LIN {X 0,Y 300.926,Z 371.519,A -85,B 0,C 180,E1 -19127.821,E2 -19127.821} C_VEL
LIN {X 0,Y 293.445,Z 384.523,A -85,B 0,C 180,E1 -19129.259,E2 -19129.259} C_VEL
LIN {X 0,Y 285.391,Z 397.595,A -85,B 0,C 180,E1 -19131.1,E2 -19131.1} C_VEL
LIN {X 0,Y 277.927,Z 408.98,A -85,B 0,C 180,E1 -19133.089,E2 -19133.089} C_VEL
LIN {X 0,Y 270.199,Z 420.219,A -85,B 0,C 180,E1 -19135.547,E2 -19135.547} C_VEL
LIN {X 0,Y 262.579,Z 430.974,A -85,B 0,C 180,E1 -19138.539,E2 -19138.539} C_VEL
LIN {X 0,Y 256.104,Z 439.853,A -85,B 0,C 180,E1 -19141.687,E2 -19141.687} C_VEL
LIN {X 0,Y 251.781,Z 445.833,A -85,B 0,C 180,E1 -19144.364,E2 -19144.364} C_VEL
LIN {X 0,Y 247.717,Z 451.471,A -85,B 0,C 180,E1 -19147.48,E2 -19147.48} C_VEL
LIN {X 0,Y 245.217,Z 454.914,A -85,B 0,C 180,E1 -19149.884,E2 -19149.884} C_VEL
LIN {X 0,Y 243.007,Z 458.084,A -85,B 0,C 180,E1 -19152.628,E2 -19152.628} C_VEL
LIN {X 0,Y 241.525,Z 462.948,A -85,B 0,C 180,E1 -19155.68,E2 -19155.68} C_VEL
LIN {X 0,Y 240.587,Z 466.054,A -85,B 0,C 180,E1 -19158.201,E2 -19158.201} C_VEL
LIN {X 0,Y 240.006,Z 469.152,A -85,B 0,C 180,E1 -19161.581,E2 -19161.581} C_VEL
LIN {X 0,Y 239.791,Z 471.129,A -85,B 0,C 180,E1 -19165.2,E2 -19165.2} C_VEL
LIN {X 0,Y 239.847,Z 471.756,A -85,B 0,C 180,E1 -19168.321,E2 -19168.321} C_VEL
LIN {X 0,Y 239.895,Z 471.645,A -85,B 0,C 180,E1 -19170,E2 -19170} C_VEL
LIN {X 0,Y 239.802,Z 470.52,A -85,B 0,C 180,E1 -19173.36,E2 -19173.36} C_VEL
LIN {X 0,Y 239.871,Z 468.169,A -85,B 0,C 180,E1 -19176.73,E2 -19176.73} C_VEL
LIN {X 0,Y 240.17,Z 464.526,A -85,B 0,C 180,E1 -19180.112,E2 -19180.112} C_VEL
LIN {X 0,Y 241.011,Z 459.793,A -85,B 0,C 180,E1 -19183.491,E2 -19183.491} C_VEL
LIN {X 0,Y 242.828,Z 456.84,A -85,B 0,C 180,E1 -19187.237,E2 -19187.237} C_VEL
LIN {X 0,Y 245.914,Z 452.461,A -85,B 0,C 180,E1 -19190.931,E2 -19190.931} C_VEL
LIN {X 0,Y 249.577,Z 447.385,A -85,B 0,C 180,E1 -19194.099,E2 -19194.099} C_VEL
LIN {X 0,Y 254.007,Z 441.145,A -85,B 0,C 180,E1 -19197.163,E2 -19197.163} C_VEL
LIN {X 0,Y 259.413,Z 433.669,A -85,B 0,C 180,E1 -19200.079,E2 -19200.079} C_VEL
LIN {X 0,Y 266.658,Z 423.616,A -85,B 0,C 180,E1 -19203.154,E2 -19203.154} C_VEL
LIN {X 0,Y 274.949,Z 411.661,A -85,B 0,C 180,E1 -19206.009,E2 -19206.009} C_VEL
LIN {X 0,Y 283.218,Z 399.07,A -85,B 0,C 180,E1 -19208.343,E2 -19208.343} C_VEL
LIN {X 0,Y 292.329,Z 384.265,A -85,B 0,C 180,E1 -19210.475,E2 -19210.475} C_VEL
LIN {X 0,Y 300.405,Z 370.081,A -85,B 0,C 180,E1 -19212.043,E2 -19212.043} C_VEL
LIN {X 0,Y 308.472,Z 354.464,A -85,B 0,C 180,E1 -19213.364,E2 -19213.364} C_VEL
LIN {X 0,Y 315.333,Z 339.378,A -85,B 0,C 180,E1 -19214.338,E2 -19214.338} C_VEL
LIN {X 0,Y 322.129,Z 322.096,A -85,B 0,C 180,E1 -19215.191,E2 -19215.191} C_VEL
LIN {X 0,Y 323.521,Z 318.179,A -85,B 0,C 180,E1 -19215.353,E2 -19215.353} C_VEL
LIN {X 0,Y 323.563,Z 317.976,A -85,B 0,C 180,E1 -19215.539,E2 -19215.539} C_VEL
LIN {X 0,Y 317.653,Z 333.405,A -85,B 0,C 180,E1 -19216.478,E2 -19216.478} C_VEL
LIN {X 0,Y 310.672,Z 348.818,A -85,B 0,C 180,E1 -19217.701,E2 -19217.701} C_VEL
LIN {X 0,Y 302.844,Z 363.944,A -85,B 0,C 180,E1 -19219.256,E2 -19219.256} C_VEL
LIN {X 0,Y 295.502,Z 376.592,A -85,B 0,C 180,E1 -19220.931,E2 -19220.931} C_VEL
LIN {X 0,Y 287.997,Z 388.352,A -85,B 0,C 180,E1 -19222.845,E2 -19222.845} C_VEL
LIN {X 0,Y 280.124,Z 399.752,A -85,B 0,C 180,E1 -19225.196,E2 -19225.196} C_VEL
LIN {X 0,Y 273.695,Z 408.358,A -85,B 0,C 180,E1 -19227.368,E2 -19227.368} C_VEL
LIN {X 0,Y 267.129,Z 416.621,A -85,B 0,C 180,E1 -19230.009,E2 -19230.009} C_VEL
LIN {X 0,Y 261.275,Z 423.494,A -85,B 0,C 180,E1 -19232.789,E2 -19232.789} C_VEL
LIN {X 0,Y 256.163,Z 429.083,A -85,B 0,C 180,E1 -19235.699,E2 -19235.699} C_VEL
LIN {X 0,Y 251.642,Z 433.523,A -85,B 0,C 180,E1 -19238.712,E2 -19238.712} C_VEL
LIN {X 0,Y 248.08,Z 436.727,A -85,B 0,C 180,E1 -19241.843,E2 -19241.843} C_VEL
LIN {X 0,Y 245.226,Z 438.819,A -85,B 0,C 180,E1 -19245.053,E2 -19245.053} C_VEL
LIN {X 0,Y 243.131,Z 439.825,A -85,B 0,C 180,E1 -19248.326,E2 -19248.326} C_VEL
LIN {X 0,Y 241.522,Z 439.746,A -85,B 0,C 180,E1 -19251.635,E2 -19251.635} C_VEL
LIN {X 0,Y 240.629,Z 438.526,A -85,B 0,C 180,E1 -19254.974,E2 -19254.974} C_VEL
LIN {X 0,Y 240.193,Z 436.107,A -85,B 0,C 180,E1 -19258.324,E2 -19258.324} C_VEL
LIN {X 0,Y 240.07,Z 432.433,A -85,B 0,C 180,E1 -19261.678,E2 -19261.678} C_VEL
LIN {X 0,Y 240.095,Z 427.408,A -85,B 0,C 180,E1 -19265.038,E2 -19265.038} C_VEL
LIN {X 0,Y 240.395,Z 422.656,A -85,B 0,C 180,E1 -19267.56,E2 -19267.56} C_VEL
LIN {X 0,Y 240.816,Z 415.933,A -85,B 0,C 180,E1 -19270.51,E2 -19270.51} C_VEL
LIN {X 0,Y 241.661,Z 407.787,A -85,B 0,C 180,E1 -19273.454,E2 -19273.454} C_VEL
LIN {X 0,Y 242.58,Z 399.463,A -85,B 0,C 180,E1 -19275.976,E2 -19275.976} C_VEL
LIN {X 0,Y 244.039,Z 387.89,A -85,B 0,C 180,E1 -19278.905,E2 -19278.905} C_VEL
LIN {X 0,Y 245.852,Z 374.969,A -85,B 0,C 180,E1 -19281.596,E2 -19281.596} C_VEL
LIN {X 0,Y 247.613,Z 361.872,A -85,B 0,C 180,E1 -19283.858,E2 -19283.858} C_VEL
LIN {X 0,Y 249.407,Z 348.878,A -85,B 0,C 180,E1 -19285.72,E2 -19285.72} C_VEL
LIN {X 0,Y 251.213,Z 333.884,A -85,B 0,C 180,E1 -19287.492,E2 -19287.492} C_VEL
LIN {X 0,Y 252.942,Z 318.105,A -85,B 0,C 180,E1 -19288.98,E2 -19288.98} C_VEL
LIN {X 0,Y 254.311,Z 301.663,A -85,B 0,C 180,E1 -19290.174,E2 -19290.174} C_VEL
LIN {X 0,Y 255.554,Z 284.029,A -85,B 0,C 180,E1 -19291.099,E2 -19291.099} C_VEL
LIN {X 0,Y 261.943,Z 188.853,A -85,B 0,C 180,E1 -19295.144,E2 -19295.144} C_VEL
LIN {X 0,Y 247.071,Z 153.283,A -85,B 0,C 180,E1 -19298.227,E2 -19298.227} C_VEL
LIN {X 0,Y 242.059,Z 141.421,A -85,B 0,C 180,E1 -19299.345,E2 -19299.345} C_VEL
LIN {X 0,Y 241.982,Z 140.968,A -85,B 0,C 180,E1 -19299.451,E2 -19299.451} C_VEL
LIN {X 0,Y 241.902,Z 140.961,A -85,B 0,C 180,E1 -19304.21,E2 -19304.21} C_VEL
LIN {X 0,Y 241.91,Z 140.944,A -85,B 0,C 180,E1 -19308.072,E2 -19308.072} C_VEL
LIN {X 0,Y 241.985,Z 140.951,A -85,B 0,C 180,E1 -19312.417,E2 -19312.417} C_VEL
LIN {X 0,Y 241.982,Z 140.957,A -85,B 0,C 180,E1 -19316.508,E2 -19316.508} C_VEL
LIN {X 0,Y 241.979,Z 140.944,A -85,B 0,C 180,E1 -19320.613,E2 -19320.613} C_VEL
LIN {X 0,Y 241.999,Z 140.959,A -85,B 0,C 180,E1 -19324.197,E2 -19324.197} C_VEL
LIN {X 0,Y 241.98,Z 141.039,A -85,B 0,C 180,E1 -19327.592,E2 -19327.592} C_VEL
LIN {X 0,Y 242.401,Z 142.66,A -85,B 0,C 180,E1 -19328.094,E2 -19328.094} C_VEL
LIN {X 0,Y 244.421,Z 146.942,A -85,B 0,C 180,E1 -19329.518,E2 -19329.518} C_VEL
LIN {X 0,Y 252.986,Z 160.771,A -85,B 0,C 180,E1 -19331.795,E2 -19331.795} C_VEL
LIN {X 0,Y 261.458,Z 175.871,A -85,B 0,C 180,E1 -19333.915,E2 -19333.915} C_VEL
LIN {X 0,Y 269.699,Z 192.53,A -85,B 0,C 180,E1 -19335.885,E2 -19335.885} C_VEL
LIN {X 0,Y 275.294,Z 205.581,A -85,B 0,C 180,E1 -19337.192,E2 -19337.192} C_VEL
LIN {X 0,Y 269.954,Z 313.697,A -85,B 0,C 180,E1 -19340.021,E2 -19340.021} C_VEL
LIN {X 0,Y 268.503,Z 329.395,A -85,B 0,C 180,E1 -19340.68,E2 -19340.68} C_VEL
LIN {X 0,Y 266.769,Z 343.814,A -85,B 0,C 180,E1 -19341.573,E2 -19341.573} C_VEL
LIN {X 0,Y 264.506,Z 358.15,A -85,B 0,C 180,E1 -19342.749,E2 -19342.749} C_VEL
LIN {X 0,Y 261.843,Z 371.771,A -85,B 0,C 180,E1 -19344.172,E2 -19344.172} C_VEL
LIN {X 0,Y 258.88,Z 385.03,A -85,B 0,C 180,E1 -19345.913,E2 -19345.913} C_VEL
LIN {X 0,Y 255.933,Z 396.923,A -85,B 0,C 180,E1 -19347.836,E2 -19347.836} C_VEL
LIN {X 0,Y 252.994,Z 407.937,A -85,B 0,C 180,E1 -19350,E2 -19350} C_VEL
LIN {X 0,Y 250.073,Z 418.104,A -85,B 0,C 180,E1 -19352.416,E2 -19352.416} C_VEL
LIN {X 0,Y 247.562,Z 426.707,A -85,B 0,C 180,E1 -19354.886,E2 -19354.886} C_VEL
LIN {X 0,Y 245.125,Z 435.113,A -85,B 0,C 180,E1 -19357.827,E2 -19357.827} C_VEL
LIN {X 0,Y 243.215,Z 441.844,A -85,B 0,C 180,E1 -19360.74,E2 -19360.74} C_VEL
LIN {X 0,Y 241.894,Z 446.911,A -85,B 0,C 180,E1 -19363.44,E2 -19363.44} C_VEL
LIN {X 0,Y 240.686,Z 452.108,A -85,B 0,C 180,E1 -19366.978,E2 -19366.978} C_VEL
LIN {X 0,Y 239.819,Z 455.891,A -85,B 0,C 180,E1 -19370.589,E2 -19370.589} C_VEL
LIN {X 0,Y 239.462,Z 458.272,A -85,B 0,C 180,E1 -19374.261,E2 -19374.261} C_VEL
LIN {X 0,Y 239.408,Z 459.268,A -85,B 0,C 180,E1 -19378.014,E2 -19378.014} C_VEL
LIN {X 0,Y 239.683,Z 458.815,A -85,B 0,C 180,E1 -19381.857,E2 -19381.857} C_VEL
LIN {X 0,Y 240.458,Z 456.825,A -85,B 0,C 180,E1 -19385.771,E2 -19385.771} C_VEL
LIN {X 0,Y 241.248,Z 454.814,A -85,B 0,C 180,E1 -19388.134,E2 -19388.134} C_VEL
LIN {X 0,Y 242.842,Z 450.587,A -85,B 0,C 180,E1 -19391.731,E2 -19391.731} C_VEL
LIN {X 0,Y 244.71,Z 445.781,A -85,B 0,C 180,E1 -19394.779,E2 -19394.779} C_VEL
LIN {X 0,Y 247.458,Z 438.873,A -85,B 0,C 180,E1 -19398.147,E2 -19398.147} C_VEL
LIN {X 0,Y 250.65,Z 431.232,A -85,B 0,C 180,E1 -19401.086,E2 -19401.086} C_VEL
LIN {X 0,Y 254.215,Z 422.206,A -85,B 0,C 180,E1 -19403.888,E2 -19403.888} C_VEL
LIN {X 0,Y 258.092,Z 411.8,A -85,B 0,C 180,E1 -19406.497,E2 -19406.497} C_VEL
LIN {X 0,Y 262.065,Z 400.682,A -85,B 0,C 180,E1 -19408.74,E2 -19408.74} C_VEL
LIN {X 0,Y 265.88,Z 388.642,A -85,B 0,C 180,E1 -19410.726,E2 -19410.726} C_VEL
LIN {X 0,Y 269.557,Z 375.766,A -85,B 0,C 180,E1 -19412.432,E2 -19412.432} C_VEL
LIN {X 0,Y 270.028,Z 373.954,A -85,B 0,C 180,E1 -19412.644,E2 -19412.644} C_VEL
LIN {X 0,Y 269.51,Z 373.561,A -85,B 0,C 180,E1 -19412.806,E2 -19412.806} C_VEL
LIN {X 0,Y 260.352,Z 374.742,A -85,B 0,C 180,E1 -19414.411,E2 -19414.411} C_VEL
LIN {X 0,Y 254.665,Z 374.937,A -85,B 0,C 180,E1 -19415.603,E2 -19415.603} C_VEL
LIN {X 0,Y 247.238,Z 374.53,A -85,B 0,C 180,E1 -19417.433,E2 -19417.433} C_VEL
LIN {X 0,Y 246.295,Z 373.126,A -85,B 0,C 180,E1 -19418.005,E2 -19418.005} C_VEL
LIN {X 0,Y 244.695,Z 384.518,A -85,B 0,C 180,E1 -19420.276,E2 -19420.276} C_VEL
LIN {X 0,Y 243.165,Z 395.558,A -85,B 0,C 180,E1 -19422.892,E2 -19422.892} C_VEL
LIN {X 0,Y 242.388,Z 402.645,A -85,B 0,C 180,E1 -19424.843,E2 -19424.843} C_VEL
LIN {X 0,Y 241.37,Z 406.257,A -85,B 0,C 180,E1 -19425.92,E2 -19425.92} C_VEL
LIN {X 0,Y 237.891,Z 411.633,A -85,B 0,C 180,E1 -19427.73,E2 -19427.73} C_VEL
LIN {X 0,Y 234.449,Z 416.584,A -85,B 0,C 180,E1 -19429.662,E2 -19429.662} C_VEL
LIN {X 0,Y 233.518,Z 419.483,A -85,B 0,C 180,E1 -19430.91,E2 -19430.91} C_VEL
LIN {X 0,Y 233.1,Z 426.282,A -85,B 0,C 180,E1 -19434.244,E2 -19434.244} C_VEL
LIN {X 0,Y 233.038,Z 431.403,A -85,B 0,C 180,E1 -19437.407,E2 -19437.407} C_VEL
LIN {X 0,Y 233.02,Z 434.736,A -85,B 0,C 180,E1 -19439.999,E2 -19439.999} C_VEL
LIN {X 0,Y 233.386,Z 438.017,A -85,B 0,C 180,E1 -19443.452,E2 -19443.452} C_VEL
LIN {X 0,Y 233.983,Z 440.115,A -85,B 0,C 180,E1 -19446.9,E2 -19446.9} C_VEL
LIN {X 0,Y 235.344,Z 441.087,A -85,B 0,C 180,E1 -19450.321,E2 -19450.321} C_VEL
LIN {X 0,Y 237.262,Z 440.964,A -85,B 0,C 180,E1 -19453.707,E2 -19453.707} C_VEL
LIN {X 0,Y 239.772,Z 439.723,A -85,B 0,C 180,E1 -19457.044,E2 -19457.044} C_VEL
LIN {X 0,Y 243.236,Z 437.397,A -85,B 0,C 180,E1 -19460.287,E2 -19460.287} C_VEL
LIN {X 0,Y 247.434,Z 434.005,A -85,B 0,C 180,E1 -19463.431,E2 -19463.431} C_VEL
LIN {X 0,Y 252.482,Z 429.476,A -85,B 0,C 180,E1 -19466.447,E2 -19466.447} C_VEL
LIN {X 0,Y 259.22,Z 422.76,A -85,B 0,C 180,E1 -19469.757,E2 -19469.757} C_VEL
LIN {X 0,Y 266.506,Z 414.81,A -85,B 0,C 180,E1 -19472.724,E2 -19472.724} C_VEL
LIN {X 0,Y 274.914,Z 404.883,A -85,B 0,C 180,E1 -19475.562,E2 -19475.562} C_VEL
LIN {X 0,Y 283.036,Z 394.461,A -85,B 0,C 180,E1 -19477.92,E2 -19477.92} C_VEL
LIN {X 0,Y 291.952,Z 382.057,A -85,B 0,C 180,E1 -19480.086,E2 -19480.086} C_VEL
LIN {X 0,Y 300.223,Z 369.287,A -85,B 0,C 180,E1 -19481.848,E2 -19481.848} C_VEL
LIN {X 0,Y 307.069,Z 357.731,A -85,B 0,C 180,E1 -19483.138,E2 -19483.138} C_VEL
LIN {X 0,Y 312.933,Z 346.743,A -85,B 0,C 180,E1 -19484.124,E2 -19484.124} C_VEL
LIN {X 0,Y 313.613,Z 345.475,A -85,B 0,C 180,E1 -19484.431,E2 -19484.431} C_VEL
LIN {X 0,Y 305.164,Z 361.795,A -85,B 0,C 180,E1 -19485.556,E2 -19485.556} C_VEL
LIN {X 0,Y 296.187,Z 377.189,A -85,B 0,C 180,E1 -19486.985,E2 -19486.985} C_VEL
LIN {X 0,Y 287.36,Z 391.028,A -85,B 0,C 180,E1 -19488.674,E2 -19488.674} C_VEL
LIN {X 0,Y 278.033,Z 404.592,A -85,B 0,C 180,E1 -19490.807,E2 -19490.807} C_VEL
LIN {X 0,Y 269.529,Z 416.205,A -85,B 0,C 180,E1 -19493.15,E2 -19493.15} C_VEL
LIN {X 0,Y 261.948,Z 426.171,A -85,B 0,C 180,E1 -19495.707,E2 -19495.707} C_VEL
LIN {X 0,Y 255.106,Z 434.753,A -85,B 0,C 180,E1 -19498.437,E2 -19498.437} C_VEL
LIN {X 0,Y 249.184,Z 442.052,A -85,B 0,C 180,E1 -19501.349,E2 -19501.349} C_VEL
LIN {X 0,Y 244.279,Z 448.164,A -85,B 0,C 180,E1 -19504.434,E2 -19504.434} C_VEL
LIN {X 0,Y 240.247,Z 453.191,A -85,B 0,C 180,E1 -19507.648,E2 -19507.648} C_VEL
LIN {X 0,Y 235.865,Z 459.03,A -85,B 0,C 180,E1 -19512.664,E2 -19512.664} C_VEL
LIN {X 0,Y 234.232,Z 464.005,A -85,B 0,C 180,E1 -19516.111,E2 -19516.111} C_VEL
LIN {X 0,Y 233.179,Z 467.672,A -85,B 0,C 180,E1 -19519.581,E2 -19519.581} C_VEL
LIN {X 0,Y 232.79,Z 470.12,A -85,B 0,C 180,E1 -19523.064,E2 -19523.064} C_VEL
LIN {X 0,Y 232.682,Z 471.387,A -85,B 0,C 180,E1 -19526.537,E2 -19526.537} C_VEL
LIN {X 0,Y 232.806,Z 471.448,A -85,B 0,C 180,E1 -19530,E2 -19530} C_VEL
LIN {X 0,Y 232.708,Z 470.282,A -85,B 0,C 180,E1 -19533.463,E2 -19533.463} C_VEL
LIN {X 0,Y 232.785,Z 467.887,A -85,B 0,C 180,E1 -19536.936,E2 -19536.936} C_VEL
LIN {X 0,Y 233.116,Z 464.197,A -85,B 0,C 180,E1 -19540.422,E2 -19540.422} C_VEL
LIN {X 0,Y 233.959,Z 459.718,A -85,B 0,C 180,E1 -19543.684,E2 -19543.684} C_VEL
LIN {X 0,Y 235.834,Z 457.13,A -85,B 0,C 180,E1 -19547.52,E2 -19547.52} C_VEL
LIN {X 0,Y 239.29,Z 452.881,A -85,B 0,C 180,E1 -19551.539,E2 -19551.539} C_VEL
LIN {X 0,Y 243.126,Z 448.136,A -85,B 0,C 180,E1 -19554.781,E2 -19554.781} C_VEL
LIN {X 0,Y 247.804,Z 442.286,A -85,B 0,C 180,E1 -19557.902,E2 -19557.902} C_VEL
LIN {X 0,Y 253.449,Z 435.245,A -85,B 0,C 180,E1 -19560.864,E2 -19560.864} C_VEL
LIN {X 0,Y 260.093,Z 426.873,A -85,B 0,C 180,E1 -19563.637,E2 -19563.637} C_VEL
LIN {X 0,Y 267.58,Z 417.126,A -85,B 0,C 180,E1 -19566.225,E2 -19566.225} C_VEL
LIN {X 0,Y 274.794,Z 407.302,A -85,B 0,C 180,E1 -19568.331,E2 -19568.331} C_VEL
LIN {X 0,Y 282.677,Z 396.052,A -85,B 0,C 180,E1 -19570.272,E2 -19570.272} C_VEL
LIN {X 0,Y 291.787,Z 382.13,A -85,B 0,C 180,E1 -19572.175,E2 -19572.175} C_VEL
LIN {X 0,Y 300.368,Z 367.891,A -85,B 0,C 180,E1 -19573.649,E2 -19573.649} C_VEL
LIN {X 0,Y 308.765,Z 352.317,A -85,B 0,C 180,E1 -19574.879,E2 -19574.879} C_VEL
LIN {X 0,Y 312.951,Z 343.745,A -85,B 0,C 180,E1 -19575.419,E2 -19575.419} C_VEL
LIN {X 0,Y 313.381,Z 342.678,A -85,B 0,C 180,E1 -19575.791,E2 -19575.791} C_VEL
LIN {X 0,Y 306.429,Z 356.216,A -85,B 0,C 180,E1 -19576.975,E2 -19576.975} C_VEL
LIN {X 0,Y 298.992,Z 369.068,A -85,B 0,C 180,E1 -19578.392,E2 -19578.392} C_VEL
LIN {X 0,Y 289.686,Z 383.476,A -85,B 0,C 180,E1 -19580.444,E2 -19580.444} C_VEL
LIN {X 0,Y 282.043,Z 394.205,A -85,B 0,C 180,E1 -19582.375,E2 -19582.375} C_VEL
LIN {X 0,Y 272.96,Z 405.879,A -85,B 0,C 180,E1 -19585.049,E2 -19585.049} C_VEL
LIN {X 0,Y 265.624,Z 414.565,A -85,B 0,C 180,E1 -19587.603,E2 -19587.603} C_VEL
LIN {X 0,Y 258.219,Z 422.674,A -85,B 0,C 180,E1 -19590.666,E2 -19590.666} C_VEL
LIN {X 0,Y 251.229,Z 429.713,A -85,B 0,C 180,E1 -19594.304,E2 -19594.304} C_VEL
LIN {X 0,Y 247.459,Z 433.067,A -85,B 0,C 180,E1 -19596.572,E2 -19596.572} C_VEL
LIN {X 0,Y 243.172,Z 436.579,A -85,B 0,C 180,E1 -19599.708,E2 -19599.708} C_VEL
LIN {X 0,Y 239.77,Z 438.959,A -85,B 0,C 180,E1 -19602.956,E2 -19602.956} C_VEL
LIN {X 0,Y 237.231,Z 440.253,A -85,B 0,C 180,E1 -19606.291,E2 -19606.291} C_VEL
LIN {X 0,Y 235.256,Z 440.439,A -85,B 0,C 180,E1 -19609.675,E2 -19609.675} C_VEL
LIN {X 0,Y 233.942,Z 439.523,A -85,B 0,C 180,E1 -19613.099,E2 -19613.099} C_VEL
LIN {X 0,Y 233.335,Z 437.473,A -85,B 0,C 180,E1 -19616.547,E2 -19616.547} C_VEL
LIN {X 0,Y 233.012,Z 434.229,A -85,B 0,C 180,E1 -19620.001,E2 -19620.001} C_VEL
LIN {X 0,Y 232.99,Z 429.672,A -85,B 0,C 180,E1 -19623.459,E2 -19623.459} C_VEL
LIN {X 0,Y 233.218,Z 423.655,A -85,B 0,C 180,E1 -19626.924,E2 -19626.924} C_VEL
LIN {X 0,Y 233.659,Z 417.081,A -85,B 0,C 180,E1 -19629.96,E2 -19629.96} C_VEL
LIN {X 0,Y 234.399,Z 409.058,A -85,B 0,C 180,E1 -19632.996,E2 -19632.996} C_VEL
LIN {X 0,Y 235.309,Z 400.854,A -85,B 0,C 180,E1 -19635.594,E2 -19635.594} C_VEL
LIN {X 0,Y 236.606,Z 390.774,A -85,B 0,C 180,E1 -19638.306,E2 -19638.306} C_VEL
LIN {X 0,Y 238.205,Z 378.995,A -85,B 0,C 180,E1 -19640.962,E2 -19640.962} C_VEL
LIN {X 0,Y 239.973,Z 366.61,A -85,B 0,C 180,E1 -19643.29,E2 -19643.29} C_VEL
LIN {X 0,Y 241.849,Z 353.276,A -85,B 0,C 180,E1 -19645.381,E2 -19645.381} C_VEL
LIN {X 0,Y 243.652,Z 338.78,A -85,B 0,C 180,E1 -19647.252,E2 -19647.252} C_VEL
LIN {X 0,Y 245.472,Z 322.964,A -85,B 0,C 180,E1 -19648.891,E2 -19648.891} C_VEL
LIN {X 0,Y 247.014,Z 306.649,A -85,B 0,C 180,E1 -19650.215,E2 -19650.215} C_VEL
LIN {X 0,Y 248.289,Z 289.889,A -85,B 0,C 180,E1 -19651.222,E2 -19651.222} C_VEL
LIN {X 0,Y 255.155,Z 190.478,A -85,B 0,C 180,E1 -19655.633,E2 -19655.633} C_VEL
LIN {X 0,Y 240.998,Z 156.526,A -85,B 0,C 180,E1 -19658.644,E2 -19658.644} C_VEL
LIN {X 0,Y 234.996,Z 142.381,A -85,B 0,C 180,E1 -19660.021,E2 -19660.021} C_VEL
LIN {X 0,Y 234.92,Z 141.848,A -85,B 0,C 180,E1 -19660.074,E2 -19660.074} C_VEL
LIN {X 0,Y 234.869,Z 141.838,A -85,B 0,C 180,E1 -19664.098,E2 -19664.098} C_VEL
LIN {X 0,Y 234.856,Z 141.833,A -85,B 0,C 180,E1 -19668.826,E2 -19668.826} C_VEL
LIN {X 0,Y 234.92,Z 141.848,A -85,B 0,C 180,E1 -19671.079,E2 -19671.079} C_VEL
LIN {X 0,Y 234.927,Z 141.818,A -85,B 0,C 180,E1 -19675.361,E2 -19675.361} C_VEL
LIN {X 0,Y 234.901,Z 141.831,A -85,B 0,C 180,E1 -19679.428,E2 -19679.428} C_VEL
LIN {X 0,Y 234.944,Z 141.843,A -85,B 0,C 180,E1 -19683.821,E2 -19683.821} C_VEL
LIN {X 0,Y 234.919,Z 141.864,A -85,B 0,C 180,E1 -19686.121,E2 -19686.121} C_VEL
LIN {X 0,Y 236.857,Z 146.96,A -85,B 0,C 180,E1 -19687.836,E2 -19687.836} C_VEL
LIN {X 0,Y 241.56,Z 154.168,A -85,B 0,C 180,E1 -19689.203,E2 -19689.203} C_VEL
LIN {X 0,Y 247.297,Z 163.395,A -85,B 0,C 180,E1 -19690.785,E2 -19690.785} C_VEL
LIN {X 0,Y 253.291,Z 173.856,A -85,B 0,C 180,E1 -19692.362,E2 -19692.362} C_VEL
LIN {X 0,Y 262.068,Z 190.798,A -85,B 0,C 180,E1 -19694.564,E2 -19694.564} C_VEL
LIN {X 0,Y 267.982,Z 204.189,A -85,B 0,C 180,E1 -19696.015,E2 -19696.015} C_VEL
LIN {X 0,Y 269.486,Z 207.769,A -85,B 0,C 180,E1 -19696.377,E2 -19696.377} C_VEL
LIN {X 0,Y 263.944,Z 314.429,A -85,B 0,C 180,E1 -19699.215,E2 -19699.215} C_VEL
LIN {X 0,Y 262.482,Z 329.827,A -85,B 0,C 180,E1 -19699.88,E2 -19699.88} C_VEL
LIN {X 0,Y 260.685,Z 344.188,A -85,B 0,C 180,E1 -19700.789,E2 -19700.789} C_VEL
LIN {X 0,Y 258.331,Z 358.5,A -85,B 0,C 180,E1 -19701.985,E2 -19701.985} C_VEL
LIN {X 0,Y 255.841,Z 370.954,A -85,B 0,C 180,E1 -19703.296,E2 -19703.296} C_VEL
LIN {X 0,Y 252.829,Z 384.171,A -85,B 0,C 180,E1 -19705.037,E2 -19705.037} C_VEL
LIN {X 0,Y 249.774,Z 396.136,A -85,B 0,C 180,E1 -19706.976,E2 -19706.976} C_VEL
LIN {X 0,Y 246.858,Z 406.743,A -85,B 0,C 180,E1 -19709.063,E2 -19709.063} C_VEL
LIN {X 0,Y 243.621,Z 417.606,A -85,B 0,C 180,E1 -19711.653,E2 -19711.653} C_VEL
LIN {X 0,Y 240.572,Z 427.609,A -85,B 0,C 180,E1 -19714.608,E2 -19714.608} C_VEL
LIN {X 0,Y 238.092,Z 435.891,A -85,B 0,C 180,E1 -19717.633,E2 -19717.633} C_VEL
LIN {X 0,Y 236.075,Z 442.798,A -85,B 0,C 180,E1 -19720.757,E2 -19720.757} C_VEL
LIN {X 0,Y 234.59,Z 448.26,A -85,B 0,C 180,E1 -19723.867,E2 -19723.867} C_VEL
LIN {X 0,Y 233.891,Z 451.241,A -85,B 0,C 180,E1 -19725.939,E2 -19725.939} C_VEL
LIN {X 0,Y 232.966,Z 455.112,A -85,B 0,C 180,E1 -19729.381,E2 -19729.381} C_VEL
LIN {X 0,Y 232.402,Z 457.92,A -85,B 0,C 180,E1 -19733.149,E2 -19733.149} C_VEL
LIN {X 0,Y 232.252,Z 459.334,A -85,B 0,C 180,E1 -19736.994,E2 -19736.994} C_VEL
LIN {X 0,Y 232.341,Z 459.507,A -85,B 0,C 180,E1 -19738.946,E2 -19738.946} C_VEL
LIN {X 0,Y 232.728,Z 458.736,A -85,B 0,C 180,E1 -19742.927,E2 -19742.927} C_VEL
LIN {X 0,Y 233.304,Z 457.378,A -85,B 0,C 180,E1 -19745.575,E2 -19745.575} C_VEL
LIN {X 0,Y 234.474,Z 454.595,A -85,B 0,C 180,E1 -19749.009,E2 -19749.009} C_VEL
LIN {X 0,Y 235.784,Z 451.426,A -85,B 0,C 180,E1 -19751.825,E2 -19751.825} C_VEL
LIN {X 0,Y 237.832,Z 446.426,A -85,B 0,C 180,E1 -19755.171,E2 -19755.171} C_VEL
LIN {X 0,Y 240.432,Z 440.271,A -85,B 0,C 180,E1 -19758.351,E2 -19758.351} C_VEL
LIN {X 0,Y 244.084,Z 432.028,A -85,B 0,C 180,E1 -19761.685,E2 -19761.685} C_VEL
LIN {X 0,Y 247.876,Z 422.941,A -85,B 0,C 180,E1 -19764.602,E2 -19764.602} C_VEL
LIN {X 0,Y 251.451,Z 413.84,A -85,B 0,C 180,E1 -19766.982,E2 -19766.982} C_VEL
LIN {X 0,Y 255.497,Z 403.115,A -85,B 0,C 180,E1 -19769.272,E2 -19769.272} C_VEL
LIN {X 0,Y 259.73,Z 390.788,A -85,B 0,C 180,E1 -19771.409,E2 -19771.409} C_VEL
LIN {X 0,Y 262.719,Z 380.941,A -85,B 0,C 180,E1 -19772.81,E2 -19772.81} C_VEL
LIN {X 0,Y 262.693,Z 380.241,A -85,B 0,C 180,E1 -19772.947,E2 -19772.947} C_VEL
LIN {X 0,Y 256.756,Z 380.836,A -85,B 0,C 180,E1 -19774.026,E2 -19774.026} C_VEL
LIN {X 0,Y 251.259,Z 380.979,A -85,B 0,C 180,E1 -19775.192,E2 -19775.192} C_VEL
LIN {X 0,Y 241.168,Z 380.509,A -85,B 0,C 180,E1 -19777.738,E2 -19777.738} C_VEL
LIN {X 0,Y 239.009,Z 379.996,A -85,B 0,C 180,E1 -19778.434,E2 -19778.434} C_VEL
LIN {X 0,Y 238.368,Z 378.84,A -85,B 0,C 180,E1 -19778.94,E2 -19778.94} C_VEL
LIN {X 0,Y 236.768,Z 390.837,A -85,B 0,C 180,E1 -19781.626,E2 -19781.626} C_VEL
LIN {X 0,Y 235.425,Z 401.24,A -85,B 0,C 180,E1 -19784.414,E2 -19784.414} C_VEL
LIN {X 0,Y 234.423,Z 409.432,A -85,B 0,C 180,E1 -19787.005,E2 -19787.005} C_VEL
LIN {X 0,Y 233.677,Z 417.483,A -85,B 0,C 180,E1 -19790.041,E2 -19790.041} C_VEL
LIN {X 0,Y 233.518,Z 419.483,A -85,B 0,C 180,E1 -19790.91,E2 -19790.91} C_VEL
LIN {X 0,Y 232.656,Z 422.259,A -85,B 0,C 180,E1 -19792.173,E2 -19792.173} C_VEL
LIN {X 0,Y 229.576,Z 426.299,A -85,B 0,C 180,E1 -19794.285,E2 -19794.285} C_VEL
LIN {X 0,Y 227.07,Z 429.149,A -85,B 0,C 180,E1 -19796.05,E2 -19796.05} C_VEL
LIN {X 0,Y 226.025,Z 431.169,A -85,B 0,C 180,E1 -19797.444,E2 -19797.444} C_VEL
LIN {X 0,Y 225.95,Z 431.81,A -85,B 0,C 180,E1 -19797.918,E2 -19797.918} C_VEL
LIN {X 0,Y 226.081,Z 436.385,A -85,B 0,C 180,E1 -19801.781,E2 -19801.781} C_VEL
LIN {X 0,Y 226.536,Z 439.321,A -85,B 0,C 180,E1 -19805.34,E2 -19805.34} C_VEL
LIN {X 0,Y 227.566,Z 441.114,A -85,B 0,C 180,E1 -19808.882,E2 -19808.882} C_VEL
LIN {X 0,Y 229.294,Z 441.739,A -85,B 0,C 180,E1 -19812.389,E2 -19812.389} C_VEL
LIN {X 0,Y 231.661,Z 441.307,A -85,B 0,C 180,E1 -19815.845,E2 -19815.845} C_VEL
LIN {X 0,Y 234.818,Z 439.845,A -85,B 0,C 180,E1 -19819.221,E2 -19819.221} C_VEL
LIN {X 0,Y 238.776,Z 437.323,A -85,B 0,C 180,E1 -19822.496,E2 -19822.496} C_VEL
LIN {X 0,Y 243.736,Z 433.64,A -85,B 0,C 180,E1 -19825.627,E2 -19825.627} C_VEL
LIN {X 0,Y 249.357,Z 428.899,A -85,B 0,C 180,E1 -19828.628,E2 -19828.628} C_VEL
LIN {X 0,Y 256.819,Z 421.948,A -85,B 0,C 180,E1 -19831.928,E2 -19831.928} C_VEL
LIN {X 0,Y 264.812,Z 413.855,A -85,B 0,C 180,E1 -19834.792,E2 -19834.792} C_VEL
LIN {X 0,Y 272.849,Z 405.006,A -85,B 0,C 180,E1 -19837.251,E2 -19837.251} C_VEL
LIN {X 0,Y 281.508,Z 394.646,A -85,B 0,C 180,E1 -19839.54,E2 -19839.54} C_VEL
LIN {X 0,Y 290.931,Z 382.32,A -85,B 0,C 180,E1 -19841.629,E2 -19841.629} C_VEL
LIN {X 0,Y 299.644,Z 369.727,A -85,B 0,C 180,E1 -19843.317,E2 -19843.317} C_VEL
LIN {X 0,Y 303.538,Z 363.662,A -85,B 0,C 180,E1 -19843.996,E2 -19843.996} C_VEL
LIN {X 0,Y 304.103,Z 362.778,A -85,B 0,C 180,E1 -19844.239,E2 -19844.239} C_VEL
LIN {X 0,Y 295.457,Z 376.696,A -85,B 0,C 180,E1 -19845.49,E2 -19845.49} C_VEL
LIN {X 0,Y 286.3,Z 390.137,A -85,B 0,C 180,E1 -19847.063,E2 -19847.063} C_VEL
LIN {X 0,Y 277.664,Z 401.923,A -85,B 0,C 180,E1 -19848.845,E2 -19848.845} C_VEL
LIN {X 0,Y 269.584,Z 412.274,A -85,B 0,C 180,E1 -19850.788,E2 -19850.788} C_VEL
LIN {X 0,Y 261.104,Z 422.6,A -85,B 0,C 180,E1 -19853.209,E2 -19853.209} C_VEL
LIN {X 0,Y 252.667,Z 432.475,A -85,B 0,C 180,E1 -19856.199,E2 -19856.199} C_VEL
LIN {X 0,Y 245.224,Z 440.861,A -85,B 0,C 180,E1 -19859.47,E2 -19859.47} C_VEL
LIN {X 0,Y 240.361,Z 446.255,A -85,B 0,C 180,E1 -19862.106,E2 -19862.106} C_VEL
LIN {X 0,Y 234.673,Z 452.577,A -85,B 0,C 180,E1 -19866.153,E2 -19866.153} C_VEL
LIN {X 0,Y 230.331,Z 457.259,A -85,B 0,C 180,E1 -19870.389,E2 -19870.389} C_VEL
LIN {X 0,Y 229.271,Z 458.427,A -85,B 0,C 180,E1 -19871.734,E2 -19871.734} C_VEL
LIN {X 0,Y 227.286,Z 463.976,A -85,B 0,C 180,E1 -19875.678,E2 -19875.678} C_VEL
LIN {X 0,Y 226.143,Z 467.59,A -85,B 0,C 180,E1 -19879.253,E2 -19879.253} C_VEL
LIN {X 0,Y 225.697,Z 469.99,A -85,B 0,C 180,E1 -19882.845,E2 -19882.845} C_VEL
LIN {X 0,Y 225.595,Z 471.211,A -85,B 0,C 180,E1 -19886.428,E2 -19886.428} C_VEL
LIN {X 0,Y 225.719,Z 471.246,A -85,B 0,C 180,E1 -19890,E2 -19890} C_VEL
LIN {X 0,Y 225.619,Z 470.036,A -85,B 0,C 180,E1 -19893.572,E2 -19893.572} C_VEL
LIN {X 0,Y 225.69,Z 467.59,A -85,B 0,C 180,E1 -19897.155,E2 -19897.155} C_VEL
LIN {X 0,Y 226.078,Z 463.848,A -85,B 0,C 180,E1 -19900.75,E2 -19900.75} C_VEL
LIN {X 0,Y 226.913,Z 459.586,A -85,B 0,C 180,E1 -19903.889,E2 -19903.889} C_VEL
LIN {X 0,Y 228.888,Z 457.343,A -85,B 0,C 180,E1 -19907.882,E2 -19907.882} C_VEL
LIN {X 0,Y 231.823,Z 454.226,A -85,B 0,C 180,E1 -19911.333,E2 -19911.333} C_VEL
LIN {X 0,Y 235.63,Z 450.064,A -85,B 0,C 180,E1 -19914.681,E2 -19914.681} C_VEL
LIN {X 0,Y 240.233,Z 444.883,A -85,B 0,C 180,E1 -19917.91,E2 -19917.91} C_VEL
LIN {X 0,Y 246.285,Z 438.175,A -85,B 0,C 180,E1 -19921.121,E2 -19921.121} C_VEL
LIN {X 0,Y 254.438,Z 428.923,A -85,B 0,C 180,E1 -19924.489,E2 -19924.489} C_VEL
LIN {X 0,Y 263.218,Z 418.511,A -85,B 0,C 180,E1 -19927.404,E2 -19927.404} C_VEL
LIN {X 0,Y 271.881,Z 407.687,A -85,B 0,C 180,E1 -19929.775,E2 -19929.775} C_VEL
LIN {X 0,Y 281.399,Z 395.068,A -85,B 0,C 180,E1 -19931.92,E2 -19931.92} C_VEL
LIN {X 0,Y 290.337,Z 382.299,A -85,B 0,C 180,E1 -19933.621,E2 -19933.621} C_VEL
LIN {X 0,Y 299.251,Z 368.448,A -85,B 0,C 180,E1 -19935.017,E2 -19935.017} C_VEL
LIN {X 0,Y 304.336,Z 359.866,A -85,B 0,C 180,E1 -19935.715,E2 -19935.715} C_VEL
LIN {X 0,Y 303.549,Z 361.081,A -85,B 0,C 180,E1 -19936.007,E2 -19936.007} C_VEL
LIN {X 0,Y 296.074,Z 372.865,A -85,B 0,C 180,E1 -19937.336,E2 -19937.336} C_VEL
LIN {X 0,Y 287.358,Z 385.255,A -85,B 0,C 180,E1 -19939.139,E2 -19939.139} C_VEL
LIN {X 0,Y 279.298,Z 395.721,A -85,B 0,C 180,E1 -19941.018,E2 -19941.018} C_VEL
LIN {X 0,Y 269.736,Z 407.086,A -85,B 0,C 180,E1 -19943.648,E2 -19943.648} C_VEL
LIN {X 0,Y 262.839,Z 414.61,A -85,B 0,C 180,E1 -19945.84,E2 -19945.84} C_VEL
LIN {X 0,Y 255.713,Z 421.867,A -85,B 0,C 180,E1 -19948.521,E2 -19948.521} C_VEL
LIN {X 0,Y 249.355,Z 427.863,A -85,B 0,C 180,E1 -19951.371,E2 -19951.371} C_VEL
LIN {X 0,Y 242.421,Z 433.729,A -85,B 0,C 180,E1 -19955.143,E2 -19955.143} C_VEL
LIN {X 0,Y 238.762,Z 436.457,A -85,B 0,C 180,E1 -19957.502,E2 -19957.502} C_VEL
LIN {X 0,Y 234.79,Z 439.038,A -85,B 0,C 180,E1 -19960.776,E2 -19960.776} C_VEL
LIN {X 0,Y 231.634,Z 440.566,A -85,B 0,C 180,E1 -19964.154,E2 -19964.154} C_VEL
LIN {X 0,Y 229.278,Z 441.062,A -85,B 0,C 180,E1 -19967.61,E2 -19967.61} C_VEL
LIN {X 0,Y 227.508,Z 440.484,A -85,B 0,C 180,E1 -19971.115,E2 -19971.115} C_VEL
LIN {X 0,Y 226.474,Z 438.741,A -85,B 0,C 180,E1 -19974.659,E2 -19974.659} C_VEL
LIN {X 0,Y 226.053,Z 435.849,A -85,B 0,C 180,E1 -19978.219,E2 -19978.219} C_VEL
LIN {X 0,Y 225.925,Z 431.71,A -85,B 0,C 180,E1 -19981.783,E2 -19981.783} C_VEL
LIN {X 0,Y 225.971,Z 426.18,A -85,B 0,C 180,E1 -19985.354,E2 -19985.354} C_VEL
LIN {X 0,Y 226.267,Z 421.065,A -85,B 0,C 180,E1 -19988.035,E2 -19988.035} C_VEL
LIN {X 0,Y 226.781,Z 413.799,A -85,B 0,C 180,E1 -19991.169,E2 -19991.169} C_VEL
LIN {X 0,Y 227.768,Z 405.044,A -85,B 0,C 180,E1 -19994.292,E2 -19994.292} C_VEL
LIN {X 0,Y 228.973,Z 394.481,A -85,B 0,C 180,E1 -19997.414,E2 -19997.414} C_VEL
LIN {X 0,Y 230.581,Z 382.704,A -85,B 0,C 180,E1 -20000.287,E2 -20000.287} C_VEL
LIN {X 0,Y 232.485,Z 369.761,A -85,B 0,C 180,E1 -20002.906,E2 -20002.906} C_VEL
LIN {X 0,Y 234.426,Z 355.591,A -85,B 0,C 180,E1 -20005.279,E2 -20005.279} C_VEL
LIN {X 0,Y 236.297,Z 341.539,A -85,B 0,C 180,E1 -20007.213,E2 -20007.213} C_VEL
LIN {X 0,Y 238.118,Z 326.409,A -85,B 0,C 180,E1 -20008.902,E2 -20008.902} C_VEL
LIN {X 0,Y 239.707,Z 311.019,A -85,B 0,C 180,E1 -20010.26,E2 -20010.26} C_VEL
LIN {X 0,Y 241.11,Z 293.85,A -85,B 0,C 180,E1 -20011.402,E2 -20011.402} C_VEL
LIN {X 0,Y 248.343,Z 192.122,A -85,B 0,C 180,E1 -20016.115,E2 -20016.115} C_VEL
LIN {X 0,Y 235.024,Z 159.909,A -85,B 0,C 180,E1 -20019.054,E2 -20019.054} C_VEL
LIN {X 0,Y 227.902,Z 143.077,A -85,B 0,C 180,E1 -20020.752,E2 -20020.752} C_VEL
LIN {X 0,Y 227.833,Z 142.731,A -85,B 0,C 180,E1 -20020.842,E2 -20020.842} C_VEL
LIN {X 0,Y 227.813,Z 142.698,A -85,B 0,C 180,E1 -20025.199,E2 -20025.199} C_VEL
LIN {X 0,Y 227.802,Z 142.726,A -85,B 0,C 180,E1 -20029.618,E2 -20029.618} C_VEL
LIN {X 0,Y 227.867,Z 142.692,A -85,B 0,C 180,E1 -20034.126,E2 -20034.126} C_VEL
LIN {X 0,Y 227.859,Z 142.722,A -85,B 0,C 180,E1 -20038.376,E2 -20038.376} C_VEL
LIN {X 0,Y 227.848,Z 142.718,A -85,B 0,C 180,E1 -20042.44,E2 -20042.44} C_VEL
LIN {X 0,Y 227.885,Z 142.715,A -85,B 0,C 180,E1 -20044.543,E2 -20044.543} C_VEL
LIN {X 0,Y 228.784,Z 145.388,A -85,B 0,C 180,E1 -20045.498,E2 -20045.498} C_VEL
LIN {X 0,Y 229.719,Z 147.248,A -85,B 0,C 180,E1 -20046.157,E2 -20046.157} C_VEL
LIN {X 0,Y 237.338,Z 158.993,A -85,B 0,C 180,E1 -20048.473,E2 -20048.473} C_VEL
LIN {X 0,Y 244.053,Z 169.971,A -85,B 0,C 180,E1 -20050.389,E2 -20050.389} C_VEL
LIN {X 0,Y 251.95,Z 184.394,A -85,B 0,C 180,E1 -20052.518,E2 -20052.518} C_VEL
LIN {X 0,Y 259.408,Z 199.706,A -85,B 0,C 180,E1 -20054.436,E2 -20054.436} C_VEL
LIN {X 0,Y 263.688,Z 209.807,A -85,B 0,C 180,E1 -20055.514,E2 -20055.514} C_VEL
LIN {X 0,Y 258.066,Z 314.302,A -85,B 0,C 180,E1 -20058.34,E2 -20058.34} C_VEL
LIN {X 0,Y 256.627,Z 329.42,A -85,B 0,C 180,E1 -20058.998,E2 -20058.998} C_VEL
LIN {X 0,Y 254.655,Z 344.559,A -85,B 0,C 180,E1 -20059.967,E2 -20059.967} C_VEL
LIN {X 0,Y 252.215,Z 358.841,A -85,B 0,C 180,E1 -20061.184,E2 -20061.184} C_VEL
LIN {X 0,Y 249.646,Z 371.266,A -85,B 0,C 180,E1 -20062.519,E2 -20062.519} C_VEL
LIN {X 0,Y 246.547,Z 384.449,A -85,B 0,C 180,E1 -20064.294,E2 -20064.294} C_VEL
LIN {X 0,Y 243.049,Z 397.487,A -85,B 0,C 180,E1 -20066.477,E2 -20066.477} C_VEL
LIN {X 0,Y 239.665,Z 409.186,A -85,B 0,C 180,E1 -20068.905,E2 -20068.905} C_VEL
LIN {X 0,Y 236.264,Z 420.126,A -85,B 0,C 180,E1 -20071.705,E2 -20071.705} C_VEL
LIN {X 0,Y 233.591,Z 428.49,A -85,B 0,C 180,E1 -20074.314,E2 -20074.314} C_VEL
LIN {X 0,Y 231.07,Z 436.646,A -85,B 0,C 180,E1 -20077.427,E2 -20077.427} C_VEL
LIN {X 0,Y 228.935,Z 443.679,A -85,B 0,C 180,E1 -20080.775,E2 -20080.775} C_VEL
LIN {X 0,Y 227.34,Z 449.494,A -85,B 0,C 180,E1 -20084.319,E2 -20084.319} C_VEL
LIN {X 0,Y 226.148,Z 454.135,A -85,B 0,C 180,E1 -20088.106,E2 -20088.106} C_VEL
LIN {X 0,Y 225.404,Z 457.368,A -85,B 0,C 180,E1 -20091.972,E2 -20091.972} C_VEL
LIN {X 0,Y 225.166,Z 459.207,A -85,B 0,C 180,E1 -20095.911,E2 -20095.911} C_VEL
LIN {X 0,Y 225.258,Z 459.697,A -85,B 0,C 180,E1 -20099.119,E2 -20099.119} C_VEL
LIN {X 0,Y 225.622,Z 459.115,A -85,B 0,C 180,E1 -20102.749,E2 -20102.749} C_VEL
LIN {X 0,Y 226.374,Z 457.448,A -85,B 0,C 180,E1 -20106.176,E2 -20106.176} C_VEL
LIN {X 0,Y 227.533,Z 454.856,A -85,B 0,C 180,E1 -20109.448,E2 -20109.448} C_VEL
LIN {X 0,Y 229.051,Z 451.421,A -85,B 0,C 180,E1 -20112.574,E2 -20112.574} C_VEL
LIN {X 0,Y 230.966,Z 447.058,A -85,B 0,C 180,E1 -20115.583,E2 -20115.583} C_VEL
LIN {X 0,Y 233.62,Z 441.179,A -85,B 0,C 180,E1 -20118.77,E2 -20118.77} C_VEL
LIN {X 0,Y 237.168,Z 433.575,A -85,B 0,C 180,E1 -20122.013,E2 -20122.013} C_VEL
LIN {X 0,Y 240.792,Z 425.427,A -85,B 0,C 180,E1 -20124.809,E2 -20124.809} C_VEL
LIN {X 0,Y 244.796,Z 415.956,A -85,B 0,C 180,E1 -20127.456,E2 -20127.456} C_VEL
LIN {X 0,Y 248.898,Z 405.715,A -85,B 0,C 180,E1 -20129.777,E2 -20129.777} C_VEL
LIN {X 0,Y 253.192,Z 393.971,A -85,B 0,C 180,E1 -20131.941,E2 -20131.941} C_VEL
LIN {X 0,Y 255.325,Z 387.59,A -85,B 0,C 180,E1 -20132.941,E2 -20132.941} C_VEL
LIN {X 0,Y 255.072,Z 386.676,A -85,B 0,C 180,E1 -20133.188,E2 -20133.188} C_VEL
LIN {X 0,Y 247.482,Z 386.842,A -85,B 0,C 180,E1 -20134.787,E2 -20134.787} C_VEL
LIN {X 0,Y 237.429,Z 386.315,A -85,B 0,C 180,E1 -20137.368,E2 -20137.368} C_VEL
LIN {X 0,Y 234.327,Z 385.588,A -85,B 0,C 180,E1 -20138.398,E2 -20138.398} C_VEL
LIN {X 0,Y 232.883,Z 385.727,A -85,B 0,C 180,E1 -20138.768,E2 -20138.768} C_VEL
LIN {X 0,Y 230.994,Z 384.912,A -85,B 0,C 180,E1 -20139.519,E2 -20139.519} C_VEL
LIN {X 0,Y 230.637,Z 383.902,A -85,B 0,C 180,E1 -20139.893,E2 -20139.893} C_VEL
LIN {X 0,Y 229.072,Z 394.904,A -85,B 0,C 180,E1 -20142.594,E2 -20142.594} C_VEL
LIN {X 0,Y 227.829,Z 405.442,A -85,B 0,C 180,E1 -20145.712,E2 -20145.712} C_VEL
LIN {X 0,Y 226.823,Z 414.209,A -85,B 0,C 180,E1 -20148.833,E2 -20148.833} C_VEL
LIN {X 0,Y 226.267,Z 421.511,A -85,B 0,C 180,E1 -20151.965,E2 -20151.965} C_VEL
LIN {X 0,Y 225.938,Z 427.562,A -85,B 0,C 180,E1 -20155.158,E2 -20155.158} C_VEL
LIN {X 0,Y 225.95,Z 431.81,A -85,B 0,C 180,E1 -20157.918,E2 -20157.918} C_VEL
LIN {X 0,Y 225.319,Z 433.662,A -85,B 0,C 180,E1 -20159.333,E2 -20159.333} C_VEL
LIN {X 0,Y 222.563,Z 436.277,A -85,B 0,C 180,E1 -20161.676,E2 -20161.676} C_VEL
LIN {X 0,Y 220.309,Z 438.006,A -85,B 0,C 180,E1 -20163.612,E2 -20163.612} C_VEL
LIN {X 0,Y 219.479,Z 439.106,A -85,B 0,C 180,E1 -20165.123,E2 -20165.123} C_VEL
LIN {X 0,Y 219.484,Z 439.434,A -85,B 0,C 180,E1 -20165.634,E2 -20165.634} C_VEL
LIN {X 0,Y 220.548,Z 441.355,A -85,B 0,C 180,E1 -20169.167,E2 -20169.167} C_VEL
LIN {X 0,Y 222.378,Z 442.272,A -85,B 0,C 180,E1 -20172.781,E2 -20172.781} C_VEL
LIN {X 0,Y 224.877,Z 442.155,A -85,B 0,C 180,E1 -20176.336,E2 -20176.336} C_VEL
LIN {X 0,Y 228.21,Z 440.943,A -85,B 0,C 180,E1 -20179.801,E2 -20179.801} C_VEL
LIN {X 0,Y 232.357,Z 438.709,A -85,B 0,C 180,E1 -20183.154,E2 -20183.154} C_VEL
LIN {X 0,Y 237.565,Z 435.405,A -85,B 0,C 180,E1 -20186.343,E2 -20186.343} C_VEL
LIN {X 0,Y 243.441,Z 431.077,A -85,B 0,C 180,E1 -20189.391,E2 -20189.391} C_VEL
LIN {X 0,Y 251.232,Z 424.609,A -85,B 0,C 180,E1 -20192.725,E2 -20192.725} C_VEL
LIN {X 0,Y 259.513,Z 417.063,A -85,B 0,C 180,E1 -20195.609,E2 -20195.609} C_VEL
LIN {X 0,Y 268.861,Z 407.705,A -85,B 0,C 180,E1 -20198.354,E2 -20198.354} C_VEL
LIN {X 0,Y 277.947,Z 397.778,A -85,B 0,C 180,E1 -20200.624,E2 -20200.624} C_VEL
LIN {X 0,Y 287.739,Z 386.068,A -85,B 0,C 180,E1 -20202.671,E2 -20202.671} C_VEL
LIN {X 0,Y 294.158,Z 377.766,A -85,B 0,C 180,E1 -20203.857,E2 -20203.857} C_VEL
LIN {X 0,Y 293.938,Z 378.156,A -85,B 0,C 180,E1 -20204.168,E2 -20204.168} C_VEL
LIN {X 0,Y 284.397,Z 391.173,A -85,B 0,C 180,E1 -20205.675,E2 -20205.675} C_VEL
LIN {X 0,Y 275.229,Z 402.719,A -85,B 0,C 180,E1 -20207.415,E2 -20207.415} C_VEL
LIN {X 0,Y 266.76,Z 412.735,A -85,B 0,C 180,E1 -20209.303,E2 -20209.303} C_VEL
LIN {X 0,Y 257.838,Z 422.732,A -85,B 0,C 180,E1 -20211.676,E2 -20211.676} C_VEL
LIN {X 0,Y 248.863,Z 432.347,A -85,B 0,C 180,E1 -20214.625,E2 -20214.625} C_VEL
LIN {X 0,Y 241.749,Z 439.648,A -85,B 0,C 180,E1 -20217.465,E2 -20217.465} C_VEL
LIN {X 0,Y 235.599,Z 445.825,A -85,B 0,C 180,E1 -20220.515,E2 -20220.515} C_VEL
LIN {X 0,Y 229.302,Z 452.024,A -85,B 0,C 180,E1 -20224.59,E2 -20224.59} C_VEL
LIN {X 0,Y 225.245,Z 455.821,A -85,B 0,C 180,E1 -20228.012,E2 -20228.012} C_VEL
LIN {X 0,Y 222.514,Z 458.401,A -85,B 0,C 180,E1 -20231.111,E2 -20231.111} C_VEL
LIN {X 0,Y 220.764,Z 462.887,A -85,B 0,C 180,E1 -20234.3,E2 -20234.3} C_VEL
LIN {X 0,Y 219.604,Z 465.896,A -85,B 0,C 180,E1 -20237.055,E2 -20237.055} C_VEL
LIN {X 0,Y 218.81,Z 468.838,A -85,B 0,C 180,E1 -20240.759,E2 -20240.759} C_VEL
LIN {X 0,Y 218.551,Z 470.595,A -85,B 0,C 180,E1 -20244.464,E2 -20244.464} C_VEL
LIN {X 0,Y 218.566,Z 471.183,A -85,B 0,C 180,E1 -20248.157,E2 -20248.157} C_VEL
LIN {X 0,Y 218.634,Z 471.033,A -85,B 0,C 180,E1 -20250,E2 -20250} C_VEL
LIN {X 0,Y 218.517,Z 469.789,A -85,B 0,C 180,E1 -20253.688,E2 -20253.688} C_VEL
LIN {X 0,Y 218.608,Z 467.294,A -85,B 0,C 180,E1 -20257.388,E2 -20257.388} C_VEL
LIN {X 0,Y 219.058,Z 463.5,A -85,B 0,C 180,E1 -20261.099,E2 -20261.099} C_VEL
LIN {X 0,Y 219.977,Z 459.29,A -85,B 0,C 180,E1 -20264.336,E2 -20264.336} C_VEL
LIN {X 0,Y 222.1,Z 457.323,A -85,B 0,C 180,E1 -20268.447,E2 -20268.447} C_VEL
LIN {X 0,Y 225.188,Z 454.513,A -85,B 0,C 180,E1 -20271.994,E2 -20271.994} C_VEL
LIN {X 0,Y 230.352,Z 449.568,A -85,B 0,C 180,E1 -20276.257,E2 -20276.257} C_VEL
LIN {X 0,Y 235.514,Z 444.477,A -85,B 0,C 180,E1 -20279.497,E2 -20279.497} C_VEL
LIN {X 0,Y 242.149,Z 437.818,A -85,B 0,C 180,E1 -20282.747,E2 -20282.747} C_VEL
LIN {X 0,Y 250.765,Z 428.899,A -85,B 0,C 180,E1 -20286.054,E2 -20286.054} C_VEL
LIN {X 0,Y 260.062,Z 418.774,A -85,B 0,C 180,E1 -20288.926,E2 -20288.926} C_VEL
LIN {X 0,Y 269.195,Z 408.274,A -85,B 0,C 180,E1 -20291.24,E2 -20291.24} C_VEL
LIN {X 0,Y 279.146,Z 396.062,A -85,B 0,C 180,E1 -20293.32,E2 -20293.32} C_VEL
LIN {X 0,Y 288.462,Z 383.73,A -85,B 0,C 180,E1 -20294.955,E2 -20294.955} C_VEL
LIN {X 0,Y 294.091,Z 375.717,A -85,B 0,C 180,E1 -20295.801,E2 -20295.801} C_VEL
LIN {X 0,Y 294.09,Z 375.631,A -85,B 0,C 180,E1 -20296.13,E2 -20296.13} C_VEL
LIN {X 0,Y 284.02,Z 388.84,A -85,B 0,C 180,E1 -20298.079,E2 -20298.079} C_VEL
LIN {X 0,Y 275.655,Z 398.736,A -85,B 0,C 180,E1 -20299.927,E2 -20299.927} C_VEL
LIN {X 0,Y 265.672,Z 409.585,A -85,B 0,C 180,E1 -20302.524,E2 -20302.524} C_VEL
LIN {X 0,Y 257.48,Z 417.683,A -85,B 0,C 180,E1 -20305.027,E2 -20305.027} C_VEL
LIN {X 0,Y 250.056,Z 424.462,A -85,B 0,C 180,E1 -20307.724,E2 -20307.724} C_VEL
LIN {X 0,Y 243.437,Z 430.019,A -85,B 0,C 180,E1 -20310.608,E2 -20310.608} C_VEL
LIN {X 0,Y 237.533,Z 434.464,A -85,B 0,C 180,E1 -20313.653,E2 -20313.653} C_VEL
LIN {X 0,Y 232.344,Z 437.845,A -85,B 0,C 180,E1 -20316.845,E2 -20316.845} C_VEL
LIN {X 0,Y 228.182,Z 440.141,A -85,B 0,C 180,E1 -20320.197,E2 -20320.197} C_VEL
LIN {X 0,Y 224.855,Z 441.4,A -85,B 0,C 180,E1 -20323.663,E2 -20323.663} C_VEL
LIN {X 0,Y 222.348,Z 441.581,A -85,B 0,C 180,E1 -20327.218,E2 -20327.218} C_VEL
LIN {X 0,Y 220.166,Z 440.359,A -85,B 0,C 180,E1 -20331.714,E2 -20331.714} C_VEL
LIN {X 0,Y 219.403,Z 438.769,A -85,B 0,C 180,E1 -20334.486,E2 -20334.486} C_VEL
LIN {X 0,Y 218.985,Z 435.658,A -85,B 0,C 180,E1 -20338.161,E2 -20338.161} C_VEL
LIN {X 0,Y 218.831,Z 431.262,A -85,B 0,C 180,E1 -20341.841,E2 -20341.841} C_VEL
LIN {X 0,Y 218.956,Z 425.146,A -85,B 0,C 180,E1 -20345.713,E2 -20345.713} C_VEL
LIN {X 0,Y 219.381,Z 418.099,A -85,B 0,C 180,E1 -20349.218,E2 -20349.218} C_VEL
LIN {X 0,Y 220.039,Z 410.121,A -85,B 0,C 180,E1 -20352.451,E2 -20352.451} C_VEL
LIN {X 0,Y 221.137,Z 400.556,A -85,B 0,C 180,E1 -20355.673,E2 -20355.673} C_VEL
LIN {X 0,Y 222.602,Z 389.163,A -85,B 0,C 180,E1 -20358.834,E2 -20358.834} C_VEL
LIN {X 0,Y 224.327,Z 377.159,A -85,B 0,C 180,E1 -20361.6,E2 -20361.6} C_VEL
LIN {X 0,Y 226.198,Z 364.337,A -85,B 0,C 180,E1 -20364.067,E2 -20364.067} C_VEL
LIN {X 0,Y 228.238,Z 349.978,A -85,B 0,C 180,E1 -20366.347,E2 -20366.347} C_VEL
LIN {X 0,Y 230.142,Z 335.29,A -85,B 0,C 180,E1 -20368.252,E2 -20368.252} C_VEL
LIN {X 0,Y 231.957,Z 319.762,A -85,B 0,C 180,E1 -20369.871,E2 -20369.871} C_VEL
LIN {X 0,Y 233.489,Z 303.066,A -85,B 0,C 180,E1 -20371.218,E2 -20371.218} C_VEL
LIN {X 0,Y 234.871,Z 285.027,A -85,B 0,C 180,E1 -20372.272,E2 -20372.272} C_VEL
LIN {X 0,Y 241.594,Z 193.691,A -85,B 0,C 180,E1 -20376.611,E2 -20376.611} C_VEL
LIN {X 0,Y 227.651,Z 160.174,A -85,B 0,C 180,E1 -20379.791,E2 -20379.791} C_VEL
LIN {X 0,Y 220.888,Z 144.252,A -85,B 0,C 180,E1 -20381.454,E2 -20381.454} C_VEL
LIN {X 0,Y 220.777,Z 143.609,A -85,B 0,C 180,E1 -20381.553,E2 -20381.553} C_VEL
LIN {X 0,Y 220.756,Z 143.572,A -85,B 0,C 180,E1 -20385.541,E2 -20385.541} C_VEL
LIN {X 0,Y 220.783,Z 143.609,A -85,B 0,C 180,E1 -20390.458,E2 -20390.458} C_VEL
LIN {X 0,Y 220.827,Z 143.578,A -85,B 0,C 180,E1 -20392.793,E2 -20392.793} C_VEL
LIN {X 0,Y 220.815,Z 143.603,A -85,B 0,C 180,E1 -20397.243,E2 -20397.243} C_VEL
LIN {X 0,Y 220.802,Z 143.583,A -85,B 0,C 180,E1 -20401.482,E2 -20401.482} C_VEL
LIN {X 0,Y 220.833,Z 143.696,A -85,B 0,C 180,E1 -20402.863,E2 -20402.863} C_VEL
LIN {X 0,Y 222.211,Z 146.976,A -85,B 0,C 180,E1 -20404.17,E2 -20404.17} C_VEL
LIN {X 0,Y 225.271,Z 151.624,A -85,B 0,C 180,E1 -20405.231,E2 -20405.231} C_VEL
LIN {X 0,Y 233.072,Z 163.683,A -85,B 0,C 180,E1 -20407.706,E2 -20407.706} C_VEL
LIN {X 0,Y 240.998,Z 176.909,A -85,B 0,C 180,E1 -20410.039,E2 -20410.039} C_VEL
LIN {X 0,Y 248.848,Z 191.803,A -85,B 0,C 180,E1 -20412.215,E2 -20412.215} C_VEL
LIN {X 0,Y 255.745,Z 206.505,A -85,B 0,C 180,E1 -20414.05,E2 -20414.05} C_VEL
LIN {X 0,Y 257.957,Z 212.137,A -85,B 0,C 180,E1 -20414.641,E2 -20414.641} C_VEL
LIN {X 0,Y 252.204,Z 314.566,A -85,B 0,C 180,E1 -20417.452,E2 -20417.452} C_VEL
LIN {X 0,Y 250.712,Z 329.52,A -85,B 0,C 180,E1 -20418.108,E2 -20418.108} C_VEL
LIN {X 0,Y 248.681,Z 344.807,A -85,B 0,C 180,E1 -20419.106,E2 -20419.106} C_VEL
LIN {X 0,Y 246.151,Z 359.093,A -85,B 0,C 180,E1 -20420.343,E2 -20420.343} C_VEL
LIN {X 0,Y 243.139,Z 373.054,A -85,B 0,C 180,E1 -20421.899,E2 -20421.899} C_VEL
LIN {X 0,Y 239.744,Z 386.647,A -85,B 0,C 180,E1 -20423.818,E2 -20423.818} C_VEL
LIN {X 0,Y 236.355,Z 398.803,A -85,B 0,C 180,E1 -20425.95,E2 -20425.95} C_VEL
LIN {X 0,Y 233.079,Z 409.632,A -85,B 0,C 180,E1 -20428.272,E2 -20428.272} C_VEL
LIN {X 0,Y 229.867,Z 419.623,A -85,B 0,C 180,E1 -20430.876,E2 -20430.876} C_VEL
LIN {X 0,Y 226.713,Z 429.111,A -85,B 0,C 180,E1 -20433.91,E2 -20433.91} C_VEL
LIN {X 0,Y 224.053,Z 437.4,A -85,B 0,C 180,E1 -20437.208,E2 -20437.208} C_VEL
LIN {X 0,Y 221.661,Z 444.869,A -85,B 0,C 180,E1 -20440.967,E2 -20440.967} C_VEL
LIN {X 0,Y 220.055,Z 450.693,A -85,B 0,C 180,E1 -20444.803,E2 -20444.803} C_VEL
LIN {X 0,Y 218.873,Z 455.07,A -85,B 0,C 180,E1 -20448.729,E2 -20448.729} C_VEL
LIN {X 0,Y 218.449,Z 457.016,A -85,B 0,C 180,E1 -20451.092,E2 -20451.092} C_VEL
LIN {X 0,Y 218.082,Z 459.265,A -85,B 0,C 180,E1 -20455.531,E2 -20455.531} C_VEL
LIN {X 0,Y 218.197,Z 459.869,A -85,B 0,C 180,E1 -20459.58,E2 -20459.58} C_VEL
LIN {X 0,Y 218.616,Z 459.237,A -85,B 0,C 180,E1 -20463.296,E2 -20463.296} C_VEL
LIN {X 0,Y 219.657,Z 457.124,A -85,B 0,C 180,E1 -20467.439,E2 -20467.439} C_VEL
LIN {X 0,Y 220.734,Z 454.888,A -85,B 0,C 180,E1 -20470.168,E2 -20470.168} C_VEL
LIN {X 0,Y 222.707,Z 450.629,A -85,B 0,C 180,E1 -20473.968,E2 -20473.968} C_VEL
LIN {X 0,Y 225.131,Z 445.609,A -85,B 0,C 180,E1 -20477.298,E2 -20477.298} C_VEL
LIN {X 0,Y 228.577,Z 438.579,A -85,B 0,C 180,E1 -20480.896,E2 -20480.896} C_VEL
LIN {X 0,Y 232.341,Z 430.818,A -85,B 0,C 180,E1 -20484.013,E2 -20484.013} C_VEL
LIN {X 0,Y 236.621,Z 421.567,A -85,B 0,C 180,E1 -20486.983,E2 -20486.983} C_VEL
LIN {X 0,Y 240.727,Z 412.061,A -85,B 0,C 180,E1 -20489.457,E2 -20489.457} C_VEL
LIN {X 0,Y 245.122,Z 401.176,A -85,B 0,C 180,E1 -20491.755,E2 -20491.755} C_VEL
LIN {X 0,Y 247.772,Z 394.119,A -85,B 0,C 180,E1 -20493.009,E2 -20493.009} C_VEL
LIN {X 0,Y 247.179,Z 392.567,A -85,B 0,C 180,E1 -20493.519,E2 -20493.519} C_VEL
LIN {X 0,Y 238.352,Z 392.317,A -85,B 0,C 180,E1 -20495.618,E2 -20495.618} C_VEL
LIN {X 0,Y 228.917,Z 391.405,A -85,B 0,C 180,E1 -20498.382,E2 -20498.382} C_VEL
LIN {X 0,Y 224.412,Z 390.553,A -85,B 0,C 180,E1 -20499.972,E2 -20499.972} C_VEL
LIN {X 0,Y 223.1,Z 389.763,A -85,B 0,C 180,E1 -20500.621,E2 -20500.621} C_VEL
LIN {X 0,Y 222.808,Z 388.975,A -85,B 0,C 180,E1 -20501.014,E2 -20501.014} C_VEL
LIN {X 0,Y 221.402,Z 399.464,A -85,B 0,C 180,E1 -20503.873,E2 -20503.873} C_VEL
LIN {X 0,Y 220.358,Z 407.975,A -85,B 0,C 180,E1 -20506.63,E2 -20506.63} C_VEL
LIN {X 0,Y 219.554,Z 416.383,A -85,B 0,C 180,E1 -20509.859,E2 -20509.859} C_VEL
LIN {X 0,Y 219.111,Z 422.458,A -85,B 0,C 180,E1 -20512.628,E2 -20512.628} C_VEL
LIN {X 0,Y 218.86,Z 429.044,A -85,B 0,C 180,E1 -20516.317,E2 -20516.317} C_VEL
LIN {X 0,Y 218.859,Z 432.989,A -85,B 0,C 180,E1 -20519.079,E2 -20519.079} C_VEL
LIN {X 0,Y 219.013,Z 436.209,A -85,B 0,C 180,E1 -20521.838,E2 -20521.838} C_VEL
LIN {X 0,Y 219.484,Z 439.434,A -85,B 0,C 180,E1 -20525.634,E2 -20525.634} C_VEL
LIN {X 0,Y 219.168,Z 440.387,A -85,B 0,C 180,E1 -20527.157,E2 -20527.157} C_VEL
LIN {X 0,Y 217.179,Z 441.671,A -85,B 0,C 180,E1 -20529.687,E2 -20529.687} C_VEL
LIN {X 0,Y 215.742,Z 442.432,A -85,B 0,C 180,E1 -20531.749,E2 -20531.749} C_VEL
LIN {X 0,Y 215.614,Z 442.801,A -85,B 0,C 180,E1 -20533.319,E2 -20533.319} C_VEL
LIN {X 0,Y 215.864,Z 442.841,A -85,B 0,C 180,E1 -20533.838,E2 -20533.838} C_VEL
LIN {X 0,Y 218.089,Z 442.88,A -85,B 0,C 180,E1 -20536.859,E2 -20536.859} C_VEL
LIN {X 0,Y 221.628,Z 441.986,A -85,B 0,C 180,E1 -20540.415,E2 -20540.415} C_VEL
LIN {X 0,Y 225.976,Z 440.12,A -85,B 0,C 180,E1 -20543.847,E2 -20543.847} C_VEL
LIN {X 0,Y 231.422,Z 437.117,A -85,B 0,C 180,E1 -20547.099,E2 -20547.099} C_VEL
LIN {X 0,Y 237.551,Z 433.138,A -85,B 0,C 180,E1 -20550.195,E2 -20550.195} C_VEL
LIN {X 0,Y 244.461,Z 428.114,A -85,B 0,C 180,E1 -20553.108,E2 -20553.108} C_VEL
LIN {X 0,Y 252.204,Z 421.951,A -85,B 0,C 180,E1 -20555.816,E2 -20555.816} C_VEL
LIN {X 0,Y 260.663,Z 414.542,A -85,B 0,C 180,E1 -20558.325,E2 -20558.325} C_VEL
LIN {X 0,Y 270.936,Z 404.665,A -85,B 0,C 180,E1 -20560.917,E2 -20560.917} C_VEL
LIN {X 0,Y 279.518,Z 395.697,A -85,B 0,C 180,E1 -20562.755,E2 -20562.755} C_VEL
LIN {X 0,Y 284.654,Z 389.936,A -85,B 0,C 180,E1 -20563.733,E2 -20563.733} C_VEL
LIN {X 0,Y 283.84,Z 390.996,A -85,B 0,C 180,E1 -20564.106,E2 -20564.106} C_VEL
LIN {X 0,Y 274.351,Z 402.211,A -85,B 0,C 180,E1 -20565.728,E2 -20565.728} C_VEL
LIN {X 0,Y 264.158,Z 413.393,A -85,B 0,C 180,E1 -20567.795,E2 -20567.795} C_VEL
LIN {X 0,Y 253.681,Z 424.19,A -85,B 0,C 180,E1 -20570.417,E2 -20570.417} C_VEL
LIN {X 0,Y 243.311,Z 434.259,A -85,B 0,C 180,E1 -20573.691,E2 -20573.691} C_VEL
LIN {X 0,Y 235.352,Z 441.612,A -85,B 0,C 180,E1 -20576.81,E2 -20576.81} C_VEL
LIN {X 0,Y 228.024,Z 448.103,A -85,B 0,C 180,E1 -20580.453,E2 -20580.453} C_VEL
LIN {X 0,Y 222.895,Z 452.531,A -85,B 0,C 180,E1 -20583.805,E2 -20583.805} C_VEL
LIN {X 0,Y 218.65,Z 456.049,A -85,B 0,C 180,E1 -20587.312,E2 -20587.312} C_VEL
LIN {X 0,Y 215.778,Z 458.458,A -85,B 0,C 180,E1 -20590.498,E2 -20590.498} C_VEL
LIN {X 0,Y 213.859,Z 462.875,A -85,B 0,C 180,E1 -20593.78,E2 -20593.78} C_VEL
LIN {X 0,Y 212.635,Z 465.856,A -85,B 0,C 180,E1 -20596.623,E2 -20596.623} C_VEL
LIN {X 0,Y 211.762,Z 468.743,A -85,B 0,C 180,E1 -20600.448,E2 -20600.448} C_VEL
LIN {X 0,Y 211.472,Z 470.447,A -85,B 0,C 180,E1 -20604.278,E2 -20604.278} C_VEL
LIN {X 0,Y 211.464,Z 470.983,A -85,B 0,C 180,E1 -20608.095,E2 -20608.095} C_VEL
LIN {X 0,Y 211.55,Z 470.809,A -85,B 0,C 180,E1 -20610,E2 -20610} C_VEL
LIN {X 0,Y 211.435,Z 469.538,A -85,B 0,C 180,E1 -20613.812,E2 -20613.812} C_VEL
LIN {X 0,Y 211.526,Z 466.994,A -85,B 0,C 180,E1 -20617.637,E2 -20617.637} C_VEL
LIN {X 0,Y 212.028,Z 463.145,A -85,B 0,C 180,E1 -20621.471,E2 -20621.471} C_VEL
LIN {X 0,Y 212.999,Z 458.951,A -85,B 0,C 180,E1 -20624.694,E2 -20624.694} C_VEL
LIN {X 0,Y 215.315,Z 457.279,A -85,B 0,C 180,E1 -20629.051,E2 -20629.051} C_VEL
LIN {X 0,Y 218.597,Z 454.766,A -85,B 0,C 180,E1 -20632.694,E2 -20632.694} C_VEL
LIN {X 0,Y 224.032,Z 450.237,A -85,B 0,C 180,E1 -20637.057,E2 -20637.057} C_VEL
LIN {X 0,Y 229.417,Z 445.476,A -85,B 0,C 180,E1 -20640.362,E2 -20640.362} C_VEL
LIN {X 0,Y 235.901,Z 439.681,A -85,B 0,C 180,E1 -20643.47,E2 -20643.47} C_VEL
LIN {X 0,Y 243.287,Z 432.876,A -85,B 0,C 180,E1 -20646.313,E2 -20646.313} C_VEL
LIN {X 0,Y 252.663,Z 423.757,A -85,B 0,C 180,E1 -20649.258,E2 -20649.258} C_VEL
LIN {X 0,Y 263.051,Z 413.001,A -85,B 0,C 180,E1 -20651.908,E2 -20651.908} C_VEL
LIN {X 0,Y 273.142,Z 401.855,A -85,B 0,C 180,E1 -20654.005,E2 -20654.005} C_VEL
LIN {X 0,Y 283.942,Z 388.933,A -85,B 0,C 180,E1 -20655.873,E2 -20655.873} C_VEL
LIN {X 0,Y 284.651,Z 387.97,A -85,B 0,C 180,E1 -20656.266,E2 -20656.266} C_VEL
LIN {X 0,Y 274.546,Z 399.294,A -85,B 0,C 180,E1 -20658.275,E2 -20658.275} C_VEL
LIN {X 0,Y 263.998,Z 410.011,A -85,B 0,C 180,E1 -20660.784,E2 -20660.784} C_VEL
LIN {X 0,Y 254.186,Z 418.954,A -85,B 0,C 180,E1 -20663.527,E2 -20663.527} C_VEL
LIN {X 0,Y 244.437,Z 426.989,A -85,B 0,C 180,E1 -20666.888,E2 -20666.888} C_VEL
LIN {X 0,Y 237.546,Z 432.113,A -85,B 0,C 180,E1 -20669.805,E2 -20669.805} C_VEL
LIN {X 0,Y 231.382,Z 436.192,A -85,B 0,C 180,E1 -20672.896,E2 -20672.896} C_VEL
LIN {X 0,Y 225.959,Z 439.232,A -85,B 0,C 180,E1 -20676.151,E2 -20676.151} C_VEL
LIN {X 0,Y 221.599,Z 441.176,A -85,B 0,C 180,E1 -20679.583,E2 -20679.583} C_VEL
LIN {X 0,Y 218.07,Z 442.134,A -85,B 0,C 180,E1 -20683.139,E2 -20683.139} C_VEL
LIN {X 0,Y 215.43,Z 442.086,A -85,B 0,C 180,E1 -20686.8,E2 -20686.8} C_VEL
LIN {X 0,Y 213.502,Z 440.933,A -85,B 0,C 180,E1 -20690.527,E2 -20690.527} C_VEL
LIN {X 0,Y 212.338,Z 438.697,A -85,B 0,C 180,E1 -20694.302,E2 -20694.302} C_VEL
LIN {X 0,Y 211.92,Z 435.323,A -85,B 0,C 180,E1 -20698.1,E2 -20698.1} C_VEL
LIN {X 0,Y 211.764,Z 430.683,A -85,B 0,C 180,E1 -20701.902,E2 -20701.902} C_VEL
LIN {X 0,Y 211.892,Z 424.619,A -85,B 0,C 180,E1 -20705.711,E2 -20705.711} C_VEL
LIN {X 0,Y 212.346,Z 416.911,A -85,B 0,C 180,E1 -20709.526,E2 -20709.526} C_VEL
LIN {X 0,Y 213.071,Z 408.644,A -85,B 0,C 180,E1 -20712.865,E2 -20712.865} C_VEL
LIN {X 0,Y 214.072,Z 400.252,A -85,B 0,C 180,E1 -20715.715,E2 -20715.715} C_VEL
LIN {X 0,Y 215.377,Z 390.057,A -85,B 0,C 180,E1 -20718.644,E2 -20718.644} C_VEL
LIN {X 0,Y 217.138,Z 377.702,A -85,B 0,C 180,E1 -20721.603,E2 -20721.603} C_VEL
LIN {X 0,Y 219.037,Z 364.909,A -85,B 0,C 180,E1 -20724.149,E2 -20724.149} C_VEL
LIN {X 0,Y 221.187,Z 350.044,A -85,B 0,C 180,E1 -20726.586,E2 -20726.586} C_VEL
LIN {X 0,Y 223.039,Z 336.047,A -85,B 0,C 180,E1 -20728.464,E2 -20728.464} C_VEL
LIN {X 0,Y 224.897,Z 320.704,A -85,B 0,C 180,E1 -20730.13,E2 -20730.13} C_VEL
LIN {X 0,Y 226.464,Z 304.394,A -85,B 0,C 180,E1 -20731.516,E2 -20731.516} C_VEL
LIN {X 0,Y 227.855,Z 286.752,A -85,B 0,C 180,E1 -20732.603,E2 -20732.603} C_VEL
LIN {X 0,Y 234.792,Z 195.235,A -85,B 0,C 180,E1 -20737.135,E2 -20737.135} C_VEL
LIN {X 0,Y 219.966,Z 159.556,A -85,B 0,C 180,E1 -20740.639,E2 -20740.639} C_VEL
LIN {X 0,Y 213.822,Z 145.137,A -85,B 0,C 180,E1 -20742.22,E2 -20742.22} C_VEL
LIN {X 0,Y 213.72,Z 144.489,A -85,B 0,C 180,E1 -20742.314,E2 -20742.314} C_VEL
LIN {X 0,Y 213.703,Z 144.445,A -85,B 0,C 180,E1 -20746.346,E2 -20746.346} C_VEL
LIN {X 0,Y 213.707,Z 144.488,A -85,B 0,C 180,E1 -20751.33,E2 -20751.33} C_VEL
LIN {X 0,Y 213.756,Z 144.46,A -85,B 0,C 180,E1 -20756.018,E2 -20756.018} C_VEL
LIN {X 0,Y 213.744,Z 144.459,A -85,B 0,C 180,E1 -20760.718,E2 -20760.718} C_VEL
LIN {X 0,Y 213.76,Z 144.56,A -85,B 0,C 180,E1 -20760.99,E2 -20760.99} C_VEL
LIN {X 0,Y 214.899,Z 147.481,A -85,B 0,C 180,E1 -20762.133,E2 -20762.133} C_VEL
LIN {X 0,Y 219.268,Z 153.744,A -85,B 0,C 180,E1 -20763.705,E2 -20763.705} C_VEL
LIN {X 0,Y 226.725,Z 164.955,A -85,B 0,C 180,E1 -20766.236,E2 -20766.236} C_VEL
LIN {X 0,Y 235.596,Z 179.747,A -85,B 0,C 180,E1 -20768.986,E2 -20768.986} C_VEL
LIN {X 0,Y 243.3,Z 194.362,A -85,B 0,C 180,E1 -20771.233,E2 -20771.233} C_VEL
LIN {X 0,Y 249.701,Z 207.894,A -85,B 0,C 180,E1 -20773.005,E2 -20773.005} C_VEL
LIN {X 0,Y 252.233,Z 214.372,A -85,B 0,C 180,E1 -20773.718,E2 -20773.718} C_VEL
LIN {X 0,Y 246.327,Z 315.393,A -85,B 0,C 180,E1 -20776.543,E2 -20776.543} C_VEL
LIN {X 0,Y 244.752,Z 330.519,A -85,B 0,C 180,E1 -20777.234,E2 -20777.234} C_VEL
LIN {X 0,Y 242.763,Z 344.903,A -85,B 0,C 180,E1 -20778.193,E2 -20778.193} C_VEL
LIN {X 0,Y 240.144,Z 359.282,A -85,B 0,C 180,E1 -20779.461,E2 -20779.461} C_VEL
LIN {X 0,Y 237.013,Z 373.259,A -85,B 0,C 180,E1 -20781.044,E2 -20781.044} C_VEL
LIN {X 0,Y 233.738,Z 385.996,A -85,B 0,C 180,E1 -20782.863,E2 -20782.863} C_VEL
LIN {X 0,Y 230.337,Z 397.928,A -85,B 0,C 180,E1 -20784.967,E2 -20784.967} C_VEL
LIN {X 0,Y 226.908,Z 408.929,A -85,B 0,C 180,E1 -20787.337,E2 -20787.337} C_VEL
LIN {X 0,Y 223.52,Z 419.071,A -85,B 0,C 180,E1 -20790,E2 -20790} C_VEL
LIN {X 0,Y 220.123,Z 428.932,A -85,B 0,C 180,E1 -20793.203,E2 -20793.203} C_VEL
LIN {X 0,Y 217.355,Z 437.09,A -85,B 0,C 180,E1 -20796.498,E2 -20796.498} C_VEL
LIN {X 0,Y 215.001,Z 444.152,A -85,B 0,C 180,E1 -20800.071,E2 -20800.071} C_VEL
LIN {X 0,Y 213.48,Z 449.269,A -85,B 0,C 180,E1 -20803.323,E2 -20803.323} C_VEL
LIN {X 0,Y 212.149,Z 454.068,A -85,B 0,C 180,E1 -20807.347,E2 -20807.347} C_VEL
LIN {X 0,Y 211.281,Z 457.462,A -85,B 0,C 180,E1 -20811.463,E2 -20811.463} C_VEL
LIN {X 0,Y 211,Z 459.458,A -85,B 0,C 180,E1 -20815.658,E2 -20815.658} C_VEL
LIN {X 0,Y 211.113,Z 460.05,A -85,B 0,C 180,E1 -20819.957,E2 -20819.957} C_VEL
LIN {X 0,Y 211.717,Z 459.157,A -85,B 0,C 180,E1 -20824.355,E2 -20824.355} C_VEL
LIN {X 0,Y 212.569,Z 457.617,A -85,B 0,C 180,E1 -20827.486,E2 -20827.486} C_VEL
LIN {X 0,Y 214.579,Z 453.716,A -85,B 0,C 180,E1 -20832.177,E2 -20832.177} C_VEL
LIN {X 0,Y 216.621,Z 449.717,A -85,B 0,C 180,E1 -20835.542,E2 -20835.542} C_VEL
LIN {X 0,Y 219.791,Z 443.568,A -85,B 0,C 180,E1 -20839.414,E2 -20839.414} C_VEL
LIN {X 0,Y 223.444,Z 436.596,A -85,B 0,C 180,E1 -20842.783,E2 -20842.783} C_VEL
LIN {X 0,Y 227.37,Z 428.814,A -85,B 0,C 180,E1 -20845.776,E2 -20845.776} C_VEL
LIN {X 0,Y 231.851,Z 419.403,A -85,B 0,C 180,E1 -20848.697,E2 -20848.697} C_VEL
LIN {X 0,Y 236.408,Z 409.277,A -85,B 0,C 180,E1 -20851.221,E2 -20851.221} C_VEL
LIN {X 0,Y 240.507,Z 399.379,A -85,B 0,C 180,E1 -20853.234,E2 -20853.234} C_VEL
LIN {X 0,Y 239.325,Z 398.079,A -85,B 0,C 180,E1 -20853.864,E2 -20853.864} C_VEL
LIN {X 0,Y 229.311,Z 397.49,A -85,B 0,C 180,E1 -20856.519,E2 -20856.519} C_VEL
LIN {X 0,Y 220.505,Z 396.157,A -85,B 0,C 180,E1 -20859.476,E2 -20859.476} C_VEL
LIN {X 0,Y 216.636,Z 395.176,A -85,B 0,C 180,E1 -20861.069,E2 -20861.069} C_VEL
LIN {X 0,Y 215.172,Z 394.161,A -85,B 0,C 180,E1 -20861.923,E2 -20861.923} C_VEL
LIN {X 0,Y 215.017,Z 393.648,A -85,B 0,C 180,E1 -20862.217,E2 -20862.217} C_VEL
LIN {X 0,Y 213.815,Z 403.657,A -85,B 0,C 180,E1 -20865.241,E2 -20865.241} C_VEL
LIN {X 0,Y 212.716,Z 412.833,A -85,B 0,C 180,E1 -20868.566,E2 -20868.566} C_VEL
LIN {X 0,Y 212.21,Z 419.483,A -85,B 0,C 180,E1 -20871.429,E2 -20871.429} C_VEL
LIN {X 0,Y 211.892,Z 425.13,A -85,B 0,C 180,E1 -20874.289,E2 -20874.289} C_VEL
LIN {X 0,Y 211.823,Z 431.226,A -85,B 0,C 180,E1 -20878.098,E2 -20878.098} C_VEL
LIN {X 0,Y 211.946,Z 435.885,A -85,B 0,C 180,E1 -20881.9,E2 -20881.9} C_VEL
LIN {X 0,Y 212.4,Z 439.317,A -85,B 0,C 180,E1 -20885.728,E2 -20885.728} C_VEL
LIN {X 0,Y 213.553,Z 441.581,A -85,B 0,C 180,E1 -20889.47,E2 -20889.47} C_VEL
LIN {X 0,Y 215.459,Z 442.781,A -85,B 0,C 180,E1 -20893.198,E2 -20893.198} C_VEL
LIN {X 0,Y 215.864,Z 442.841,A -85,B 0,C 180,E1 -20893.838,E2 -20893.838} C_VEL
LIN {X 0,Y 216.294,Z 443.03,A -85,B 0,C 180,E1 -20895.399,E2 -20895.399} C_VEL
LIN {X 0,Y 215.573,Z 443.181,A -85,B 0,C 180,E1 -20898.021,E2 -20898.021} C_VEL
LIN {X 0,Y 215.194,Z 443.074,A -85,B 0,C 180,E1 -20900.129,E2 -20900.129} C_VEL
LIN {X 0,Y 215.883,Z 442.775,A -85,B 0,C 180,E1 -20901.685,E2 -20901.685} C_VEL
LIN {X 0,Y 216.406,Z 442.567,A -85,B 0,C 180,E1 -20902.185,E2 -20902.185} C_VEL
LIN {X 0,Y 222.298,Z 440.231,A -85,B 0,C 180,E1 -20906.27,E2 -20906.27} C_VEL
LIN {X 0,Y 228.372,Z 437.15,A -85,B 0,C 180,E1 -20909.497,E2 -20909.497} C_VEL
LIN {X 0,Y 237.026,Z 431.837,A -85,B 0,C 180,E1 -20913.266,E2 -20913.266} C_VEL
LIN {X 0,Y 244.811,Z 426.445,A -85,B 0,C 180,E1 -20916.051,E2 -20916.051} C_VEL
LIN {X 0,Y 255.646,Z 418.01,A -85,B 0,C 180,E1 -20919.219,E2 -20919.219} C_VEL
LIN {X 0,Y 265.02,Z 409.969,A -85,B 0,C 180,E1 -20921.526,E2 -20921.526} C_VEL
LIN {X 0,Y 275.069,Z 400.508,A -85,B 0,C 180,E1 -20923.618,E2 -20923.618} C_VEL
LIN {X 0,Y 273.792,Z 401.956,A -85,B 0,C 180,E1 -20924.05,E2 -20924.05} C_VEL
LIN {X 0,Y 261.811,Z 414.167,A -85,B 0,C 180,E1 -20926.272,E2 -20926.272} C_VEL
LIN {X 0,Y 250.833,Z 424.576,A -85,B 0,C 180,E1 -20928.819,E2 -20928.819} C_VEL
LIN {X 0,Y 241.973,Z 432.543,A -85,B 0,C 180,E1 -20931.357,E2 -20931.357} C_VEL
LIN {X 0,Y 231.983,Z 440.958,A -85,B 0,C 180,E1 -20934.857,E2 -20934.857} C_VEL
LIN {X 0,Y 225.026,Z 446.499,A -85,B 0,C 180,E1 -20937.931,E2 -20937.931} C_VEL
LIN {X 0,Y 219.089,Z 451.092,A -85,B 0,C 180,E1 -20941.238,E2 -20941.238} C_VEL
LIN {X 0,Y 214.197,Z 454.752,A -85,B 0,C 180,E1 -20944.752,E2 -20944.752} C_VEL
LIN {X 0,Y 209.249,Z 458.178,A -85,B 0,C 180,E1 -20949.607,E2 -20949.607} C_VEL
LIN {X 0,Y 206.981,Z 462.881,A -85,B 0,C 180,E1 -20953.225,E2 -20953.225} C_VEL
LIN {X 0,Y 205.687,Z 465.823,A -85,B 0,C 180,E1 -20956.162,E2 -20956.162} C_VEL
LIN {X 0,Y 204.702,Z 468.649,A -85,B 0,C 180,E1 -20960.115,E2 -20960.115} C_VEL
LIN {X 0,Y 204.375,Z 470.3,A -85,B 0,C 180,E1 -20964.079,E2 -20964.079} C_VEL
LIN {X 0,Y 204.366,Z 470.782,A -85,B 0,C 180,E1 -20968.029,E2 -20968.029} C_VEL
LIN {X 0,Y 204.468,Z 470.582,A -85,B 0,C 180,E1 -20970,E2 -20970} C_VEL
LIN {X 0,Y 204.345,Z 469.152,A -85,B 0,C 180,E1 -20974.144,E2 -20974.144} C_VEL
LIN {X 0,Y 204.447,Z 466.682,A -85,B 0,C 180,E1 -20977.903,E2 -20977.903} C_VEL
LIN {X 0,Y 204.992,Z 462.774,A -85,B 0,C 180,E1 -20981.871,E2 -20981.871} C_VEL
LIN {X 0,Y 206.032,Z 458.571,A -85,B 0,C 180,E1 -20985.076,E2 -20985.076} C_VEL
LIN {X 0,Y 208.572,Z 457.167,A -85,B 0,C 180,E1 -20989.692,E2 -20989.692} C_VEL
LIN {X 0,Y 212.023,Z 454.939,A -85,B 0,C 180,E1 -20993.439,E2 -20993.439} C_VEL
LIN {X 0,Y 216.465,Z 451.796,A -85,B 0,C 180,E1 -20997.035,E2 -20997.035} C_VEL
LIN {X 0,Y 223.384,Z 446.498,A -85,B 0,C 180,E1 -21001.273,E2 -21001.273} C_VEL
LIN {X 0,Y 230.923,Z 440.461,A -85,B 0,C 180,E1 -21004.743,E2 -21004.743} C_VEL
LIN {X 0,Y 239.859,Z 432.959,A -85,B 0,C 180,E1 -21007.975,E2 -21007.975} C_VEL
LIN {X 0,Y 249.767,Z 424.138,A -85,B 0,C 180,E1 -21010.86,E2 -21010.86} C_VEL
LIN {X 0,Y 260.663,Z 413.785,A -85,B 0,C 180,E1 -21013.435,E2 -21013.435} C_VEL
LIN {X 0,Y 271.189,Z 403.034,A -85,B 0,C 180,E1 -21015.453,E2 -21015.453} C_VEL
LIN {X 0,Y 273.916,Z 400.077,A -85,B 0,C 180,E1 -21015.923,E2 -21015.923} C_VEL
LIN {X 0,Y 275.077,Z 398.741,A -85,B 0,C 180,E1 -21016.384,E2 -21016.384} C_VEL
LIN {X 0,Y 265.045,Z 408.397,A -85,B 0,C 180,E1 -21018.479,E2 -21018.479} C_VEL
LIN {X 0,Y 255.629,Z 416.644,A -85,B 0,C 180,E1 -21020.778,E2 -21020.778} C_VEL
LIN {X 0,Y 246.876,Z 423.632,A -85,B 0,C 180,E1 -21023.286,E2 -21023.286} C_VEL
LIN {X 0,Y 238.88,Z 429.469,A -85,B 0,C 180,E1 -21026.014,E2 -21026.014} C_VEL
LIN {X 0,Y 231.719,Z 434.186,A -85,B 0,C 180,E1 -21028.963,E2 -21028.963} C_VEL
LIN {X 0,Y 225.26,Z 437.854,A -85,B 0,C 180,E1 -21032.097,E2 -21032.097} C_VEL
LIN {X 0,Y 219.603,Z 440.527,A -85,B 0,C 180,E1 -21035.416,E2 -21035.416} C_VEL
LIN {X 0,Y 215.024,Z 442.19,A -85,B 0,C 180,E1 -21038.929,E2 -21038.929} C_VEL
LIN {X 0,Y 211.306,Z 442.827,A -85,B 0,C 180,E1 -21042.583,E2 -21042.583} C_VEL
LIN {X 0,Y 208.536,Z 442.452,A -85,B 0,C 180,E1 -21046.355,E2 -21046.355} C_VEL
LIN {X 0,Y 206.506,Z 441.067,A -85,B 0,C 180,E1 -21050.203,E2 -21050.203} C_VEL
LIN {X 0,Y 205.277,Z 438.6,A -85,B 0,C 180,E1 -21054.105,E2 -21054.105} C_VEL
LIN {X 0,Y 204.855,Z 434.944,A -85,B 0,C 180,E1 -21058.035,E2 -21058.035} C_VEL
LIN {X 0,Y 204.698,Z 430.021,A -85,B 0,C 180,E1 -21061.968,E2 -21061.968} C_VEL
LIN {X 0,Y 204.837,Z 423.663,A -85,B 0,C 180,E1 -21065.909,E2 -21065.909} C_VEL
LIN {X 0,Y 205.261,Z 416.743,A -85,B 0,C 180,E1 -21069.361,E2 -21069.361} C_VEL
LIN {X 0,Y 205.976,Z 408.36,A -85,B 0,C 180,E1 -21072.814,E2 -21072.814} C_VEL
LIN {X 0,Y 207.001,Z 399.863,A -85,B 0,C 180,E1 -21075.761,E2 -21075.761} C_VEL
LIN {X 0,Y 208.47,Z 388.611,A -85,B 0,C 180,E1 -21079.037,E2 -21079.037} C_VEL
LIN {X 0,Y 210.3,Z 375.954,A -85,B 0,C 180,E1 -21082.085,E2 -21082.085} C_VEL
LIN {X 0,Y 212.264,Z 362.81,A -85,B 0,C 180,E1 -21084.71,E2 -21084.71} C_VEL
LIN {X 0,Y 214.365,Z 348.588,A -85,B 0,C 180,E1 -21087.059,E2 -21087.059} C_VEL
LIN {X 0,Y 216.443,Z 332.947,A -85,B 0,C 180,E1 -21089.148,E2 -21089.148} C_VEL
LIN {X 0,Y 218.36,Z 316.662,A -85,B 0,C 180,E1 -21090.862,E2 -21090.862} C_VEL
LIN {X 0,Y 219.922,Z 299.818,A -85,B 0,C 180,E1 -21092.228,E2 -21092.228} C_VEL
LIN {X 0,Y 221.505,Z 278.647,A -85,B 0,C 180,E1 -21093.456,E2 -21093.456} C_VEL
LIN {X 0,Y 227.984,Z 196.825,A -85,B 0,C 180,E1 -21097.649,E2 -21097.649} C_VEL
LIN {X 0,Y 213.792,Z 162.528,A -85,B 0,C 180,E1 -21101.136,E2 -21101.136} C_VEL
LIN {X 0,Y 206.736,Z 145.739,A -85,B 0,C 180,E1 -21103.021,E2 -21103.021} C_VEL
LIN {X 0,Y 206.68,Z 145.362,A -85,B 0,C 180,E1 -21103.09,E2 -21103.09} C_VEL
LIN {X 0,Y 206.633,Z 145.337,A -85,B 0,C 180,E1 -21108.441,E2 -21108.441} C_VEL
LIN {X 0,Y 206.67,Z 145.347,A -85,B 0,C 180,E1 -21112.258,E2 -21112.258} C_VEL
LIN {X 0,Y 206.702,Z 145.327,A -85,B 0,C 180,E1 -21114.689,E2 -21114.689} C_VEL
LIN {X 0,Y 206.722,Z 145.406,A -85,B 0,C 180,E1 -21118.918,E2 -21118.918} C_VEL
LIN {X 0,Y 207.524,Z 147.898,A -85,B 0,C 180,E1 -21119.845,E2 -21119.845} C_VEL
LIN {X 0,Y 211.617,Z 153.298,A -85,B 0,C 180,E1 -21121.453,E2 -21121.453} C_VEL
LIN {X 0,Y 218.266,Z 163.043,A -85,B 0,C 180,E1 -21123.898,E2 -21123.898} C_VEL
LIN {X 0,Y 224.816,Z 173.43,A -85,B 0,C 180,E1 -21126.154,E2 -21126.154} C_VEL
LIN {X 0,Y 232.784,Z 187.05,A -85,B 0,C 180,E1 -21128.672,E2 -21128.672} C_VEL
LIN {X 0,Y 241.997,Z 205.489,A -85,B 0,C 180,E1 -21131.424,E2 -21131.424} C_VEL
LIN {X 0,Y 246.606,Z 216.174,A -85,B 0,C 180,E1 -21132.743,E2 -21132.743} C_VEL
LIN {X 0,Y 240.568,Z 315.618,A -85,B 0,C 180,E1 -21135.568,E2 -21135.568} C_VEL
LIN {X 0,Y 238.918,Z 330.936,A -85,B 0,C 180,E1 -21136.281,E2 -21136.281} C_VEL
LIN {X 0,Y 236.786,Z 345.697,A -85,B 0,C 180,E1 -21137.29,E2 -21137.29} C_VEL
LIN {X 0,Y 234.2,Z 359.469,A -85,B 0,C 180,E1 -21138.533,E2 -21138.533} C_VEL
LIN {X 0,Y 231.365,Z 371.894,A -85,B 0,C 180,E1 -21139.941,E2 -21139.941} C_VEL
LIN {X 0,Y 227.96,Z 384.914,A -85,B 0,C 180,E1 -21141.793,E2 -21141.793} C_VEL
LIN {X 0,Y 224.342,Z 397.074,A -85,B 0,C 180,E1 -21143.931,E2 -21143.931} C_VEL
LIN {X 0,Y 220.79,Z 408.228,A -85,B 0,C 180,E1 -21146.35,E2 -21146.35} C_VEL
LIN {X 0,Y 217.175,Z 418.666,A -85,B 0,C 180,E1 -21149.119,E2 -21149.119} C_VEL
LIN {X 0,Y 213.654,Z 428.502,A -85,B 0,C 180,E1 -21152.357,E2 -21152.357} C_VEL
LIN {X 0,Y 210.696,Z 436.776,A -85,B 0,C 180,E1 -21155.743,E2 -21155.743} C_VEL
LIN {X 0,Y 208.639,Z 442.691,A -85,B 0,C 180,E1 -21158.719,E2 -21158.719} C_VEL
LIN {X 0,Y 206.559,Z 449.119,A -85,B 0,C 180,E1 -21162.777,E2 -21162.777} C_VEL
LIN {X 0,Y 205.257,Z 453.579,A -85,B 0,C 180,E1 -21166.517,E2 -21166.517} C_VEL
LIN {X 0,Y 204.374,Z 456.73,A -85,B 0,C 180,E1 -21170.113,E2 -21170.113} C_VEL
LIN {X 0,Y 203.901,Z 459.164,A -85,B 0,C 180,E1 -21174.432,E2 -21174.432} C_VEL
LIN {X 0,Y 203.873,Z 459.859,A -85,B 0,C 180,E1 -21176.625,E2 -21176.625} C_VEL
LIN {X 0,Y 204.058,Z 460.218,A -85,B 0,C 180,E1 -21180.566,E2 -21180.566} C_VEL
LIN {X 0,Y 204.644,Z 459.457,A -85,B 0,C 180,E1 -21184.489,E2 -21184.489} C_VEL
LIN {X 0,Y 205.684,Z 457.711,A -85,B 0,C 180,E1 -21188.196,E2 -21188.196} C_VEL
LIN {X 0,Y 207.66,Z 454.195,A -85,B 0,C 180,E1 -21192.6,E2 -21192.6} C_VEL
LIN {X 0,Y 209.819,Z 450.224,A -85,B 0,C 180,E1 -21196.088,E2 -21196.088} C_VEL
LIN {X 0,Y 212.601,Z 445.149,A -85,B 0,C 180,E1 -21199.492,E2 -21199.492} C_VEL
LIN {X 0,Y 216.103,Z 438.827,A -85,B 0,C 180,E1 -21202.823,E2 -21202.823} C_VEL
LIN {X 0,Y 220.292,Z 431.133,A -85,B 0,C 180,E1 -21206.045,E2 -21206.045} C_VEL
LIN {X 0,Y 225.099,Z 421.775,A -85,B 0,C 180,E1 -21209.16,E2 -21209.16} C_VEL
LIN {X 0,Y 229.991,Z 411.516,A -85,B 0,C 180,E1 -21211.881,E2 -21211.881} C_VEL
LIN {X 0,Y 233.583,Z 403.465,A -85,B 0,C 180,E1 -21213.653,E2 -21213.653} C_VEL
LIN {X 0,Y 220.378,Z 402.23,A -85,B 0,C 180,E1 -21217.499,E2 -21217.499} C_VEL
LIN {X 0,Y 212.295,Z 400.575,A -85,B 0,C 180,E1 -21220.667,E2 -21220.667} C_VEL
LIN {X 0,Y 208.695,Z 399.604,A -85,B 0,C 180,E1 -21222.356,E2 -21222.356} C_VEL
LIN {X 0,Y 207.431,Z 398.585,A -85,B 0,C 180,E1 -21223.262,E2 -21223.262} C_VEL
LIN {X 0,Y 207.316,Z 398.19,A -85,B 0,C 180,E1 -21223.569,E2 -21223.569} C_VEL
LIN {X 0,Y 206.15,Z 407.517,A -85,B 0,C 180,E1 -21226.695,E2 -21226.695} C_VEL
LIN {X 0,Y 205.359,Z 416.139,A -85,B 0,C 180,E1 -21230.147,E2 -21230.147} C_VEL
LIN {X 0,Y 204.837,Z 424.173,A -85,B 0,C 180,E1 -21234.091,E2 -21234.091} C_VEL
LIN {X 0,Y 204.755,Z 430.57,A -85,B 0,C 180,E1 -21238.032,E2 -21238.032} C_VEL
LIN {X 0,Y 204.881,Z 435.52,A -85,B 0,C 180,E1 -21241.965,E2 -21241.965} C_VEL
LIN {X 0,Y 205.33,Z 439.213,A -85,B 0,C 180,E1 -21245.893,E2 -21245.893} C_VEL
LIN {X 0,Y 206.57,Z 441.721,A -85,B 0,C 180,E1 -21249.794,E2 -21249.794} C_VEL
LIN {X 0,Y 208.895,Z 443.246,A -85,B 0,C 180,E1 -21254.166,E2 -21254.166} C_VEL
LIN {X 0,Y 211.322,Z 443.588,A -85,B 0,C 180,E1 -21257.416,E2 -21257.416} C_VEL
LIN {X 0,Y 215.072,Z 442.997,A -85,B 0,C 180,E1 -21261.066,E2 -21261.066} C_VEL
LIN {X 0,Y 216.406,Z 442.567,A -85,B 0,C 180,E1 -21262.185,E2 -21262.185} C_VEL
LIN {X 0,Y 217.035,Z 442.29,A -85,B 0,C 180,E1 -21263.227,E2 -21263.227} C_VEL
LIN {X 0,Y 216.337,Z 441.696,A -85,B 0,C 180,E1 -21266.787,E2 -21266.787} C_VEL
LIN {X 0,Y 217.396,Z 441.135,A -85,B 0,C 180,E1 -21267.785,E2 -21267.785} C_VEL
LIN {X 0,Y 222.422,Z 438.91,A -85,B 0,C 180,E1 -21270.368,E2 -21270.368} C_VEL
LIN {X 0,Y 231.439,Z 434.119,A -85,B 0,C 180,E1 -21274.178,E2 -21274.178} C_VEL
LIN {X 0,Y 239.505,Z 429.157,A -85,B 0,C 180,E1 -21276.98,E2 -21276.98} C_VEL
LIN {X 0,Y 250.691,Z 421.407,A -85,B 0,C 180,E1 -21280.15,E2 -21280.15} C_VEL
LIN {X 0,Y 261.603,Z 412.929,A -85,B 0,C 180,E1 -21282.714,E2 -21282.714} C_VEL
LIN {X 0,Y 265.403,Z 409.756,A -85,B 0,C 180,E1 -21283.51,E2 -21283.51} C_VEL
LIN {X 0,Y 263.767,Z 411.359,A -85,B 0,C 180,E1 -21283.994,E2 -21283.994} C_VEL
LIN {X 0,Y 253.223,Z 420.829,A -85,B 0,C 180,E1 -21286.064,E2 -21286.064} C_VEL
LIN {X 0,Y 243.409,Z 429.085,A -85,B 0,C 180,E1 -21288.388,E2 -21288.388} C_VEL
LIN {X 0,Y 232.357,Z 437.825,A -85,B 0,C 180,E1 -21291.68,E2 -21291.68} C_VEL
LIN {X 0,Y 222.564,Z 445.022,A -85,B 0,C 180,E1 -21295.362,E2 -21295.362} C_VEL
LIN {X 0,Y 215.884,Z 449.73,A -85,B 0,C 180,E1 -21298.609,E2 -21298.609} C_VEL
LIN {X 0,Y 210.218,Z 453.448,A -85,B 0,C 180,E1 -21302.092,E2 -21302.092} C_VEL
LIN {X 0,Y 205.56,Z 456.311,A -85,B 0,C 180,E1 -21305.778,E2 -21305.778} C_VEL
LIN {X 0,Y 202.766,Z 457.899,A -85,B 0,C 180,E1 -21308.658,E2 -21308.658} C_VEL
LIN {X 0,Y 200.133,Z 462.892,A -85,B 0,C 180,E1 -21312.633,E2 -21312.633} C_VEL
LIN {X 0,Y 198.759,Z 465.803,A -85,B 0,C 180,E1 -21315.669,E2 -21315.669} C_VEL
LIN {X 0,Y 197.663,Z 468.564,A -85,B 0,C 180,E1 -21319.76,E2 -21319.76} C_VEL
LIN {X 0,Y 197.288,Z 470.154,A -85,B 0,C 180,E1 -21323.865,E2 -21323.865} C_VEL
LIN {X 0,Y 197.271,Z 470.581,A -85,B 0,C 180,E1 -21327.958,E2 -21327.958} C_VEL
LIN {X 0,Y 197.369,Z 470.354,A -85,B 0,C 180,E1 -21330,E2 -21330} C_VEL
LIN {X 0,Y 197.247,Z 468.983,A -85,B 0,C 180,E1 -21334.086,E2 -21334.086} C_VEL
LIN {X 0,Y 197.388,Z 466.359,A -85,B 0,C 180,E1 -21338.188,E2 -21338.188} C_VEL
LIN {X 0,Y 197.976,Z 462.401,A -85,B 0,C 180,E1 -21342.298,E2 -21342.298} C_VEL
LIN {X 0,Y 199.18,Z 458.031,A -85,B 0,C 180,E1 -21345.739,E2 -21345.739} C_VEL
LIN {X 0,Y 201.85,Z 456.987,A -85,B 0,C 180,E1 -21350.376,E2 -21350.376} C_VEL
LIN {X 0,Y 205.502,Z 455.076,A -85,B 0,C 180,E1 -21354.229,E2 -21354.229} C_VEL
LIN {X 0,Y 210.145,Z 452.206,A -85,B 0,C 180,E1 -21357.918,E2 -21357.918} C_VEL
LIN {X 0,Y 215.786,Z 448.492,A -85,B 0,C 180,E1 -21361.407,E2 -21361.407} C_VEL
LIN {X 0,Y 224.381,Z 442.466,A -85,B 0,C 180,E1 -21365.413,E2 -21365.413} C_VEL
LIN {X 0,Y 232.344,Z 436.518,A -85,B 0,C 180,E1 -21368.323,E2 -21368.323} C_VEL
LIN {X 0,Y 241.173,Z 429.562,A -85,B 0,C 180,E1 -21370.971,E2 -21370.971} C_VEL
LIN {X 0,Y 252.034,Z 420.425,A -85,B 0,C 180,E1 -21373.643,E2 -21373.643} C_VEL
LIN {X 0,Y 262.528,Z 410.978,A -85,B 0,C 180,E1 -21375.734,E2 -21375.734} C_VEL
LIN {X 0,Y 263.884,Z 409.674,A -85,B 0,C 180,E1 -21375.979,E2 -21375.979} C_VEL
LIN {X 0,Y 265.463,Z 408.125,A -85,B 0,C 180,E1 -21376.502,E2 -21376.502} C_VEL
LIN {X 0,Y 255.429,Z 416.427,A -85,B 0,C 180,E1 -21378.674,E2 -21378.674} C_VEL
LIN {X 0,Y 246.04,Z 423.484,A -85,B 0,C 180,E1 -21381.067,E2 -21381.067} C_VEL
LIN {X 0,Y 237.398,Z 429.347,A -85,B 0,C 180,E1 -21383.695,E2 -21383.695} C_VEL
LIN {X 0,Y 229.507,Z 434.147,A -85,B 0,C 180,E1 -21386.551,E2 -21386.551} C_VEL
LIN {X 0,Y 222.497,Z 437.917,A -85,B 0,C 180,E1 -21389.643,E2 -21389.643} C_VEL
LIN {X 0,Y 216.138,Z 440.77,A -85,B 0,C 180,E1 -21392.921,E2 -21392.921} C_VEL
LIN {X 0,Y 210.738,Z 442.556,A -85,B 0,C 180,E1 -21396.41,E2 -21396.41} C_VEL
LIN {X 0,Y 206.382,Z 443.383,A -85,B 0,C 180,E1 -21400.091,E2 -21400.091} C_VEL
LIN {X 0,Y 202.993,Z 443.262,A -85,B 0,C 180,E1 -21403.921,E2 -21403.921} C_VEL
LIN {X 0,Y 200.463,Z 442.077,A -85,B 0,C 180,E1 -21407.858,E2 -21407.858} C_VEL
LIN {X 0,Y 198.687,Z 439.723,A -85,B 0,C 180,E1 -21412.065,E2 -21412.065} C_VEL
LIN {X 0,Y 197.853,Z 435.546,A -85,B 0,C 180,E1 -21416.946,E2 -21416.946} C_VEL
LIN {X 0,Y 197.643,Z 430.688,A -85,B 0,C 180,E1 -21421.019,E2 -21421.019} C_VEL
LIN {X 0,Y 197.704,Z 424.196,A -85,B 0,C 180,E1 -21425.224,E2 -21425.224} C_VEL
LIN {X 0,Y 198.168,Z 416.516,A -85,B 0,C 180,E1 -21429.184,E2 -21429.184} C_VEL
LIN {X 0,Y 198.891,Z 408.011,A -85,B 0,C 180,E1 -21432.76,E2 -21432.76} C_VEL
LIN {X 0,Y 199.919,Z 399.399,A -85,B 0,C 180,E1 -21435.81,E2 -21435.81} C_VEL
LIN {X 0,Y 201.324,Z 388.643,A -85,B 0,C 180,E1 -21439.024,E2 -21439.024} C_VEL
LIN {X 0,Y 203.139,Z 376.286,A -85,B 0,C 180,E1 -21442.102,E2 -21442.102} C_VEL
LIN {X 0,Y 205.147,Z 363.193,A -85,B 0,C 180,E1 -21444.814,E2 -21444.814} C_VEL
LIN {X 0,Y 207.268,Z 349.007,A -85,B 0,C 180,E1 -21447.243,E2 -21447.243} C_VEL
LIN {X 0,Y 209.365,Z 333.52,A -85,B 0,C 180,E1 -21449.384,E2 -21449.384} C_VEL
LIN {X 0,Y 211.375,Z 317.267,A -85,B 0,C 180,E1 -21451.161,E2 -21451.161} C_VEL
LIN {X 0,Y 212.991,Z 299.799,A -85,B 0,C 180,E1 -21452.636,E2 -21452.636} C_VEL
LIN {X 0,Y 214.79,Z 276.831,A -85,B 0,C 180,E1 -21454.009,E2 -21454.009} C_VEL
LIN {X 0,Y 221.172,Z 198.405,A -85,B 0,C 180,E1 -21458.183,E2 -21458.183} C_VEL
LIN {X 0,Y 206.527,Z 162.941,A -85,B 0,C 180,E1 -21461.922,E2 -21461.922} C_VEL
LIN {X 0,Y 199.666,Z 146.581,A -85,B 0,C 180,E1 -21463.846,E2 -21463.846} C_VEL
LIN {X 0,Y 199.608,Z 146.227,A -85,B 0,C 180,E1 -21463.918,E2 -21463.918} C_VEL
LIN {X 0,Y 199.571,Z 146.21,A -85,B 0,C 180,E1 -21468.003,E2 -21468.003} C_VEL
LIN {X 0,Y 199.599,Z 146.249,A -85,B 0,C 180,E1 -21470.773,E2 -21470.773} C_VEL
LIN {X 0,Y 199.613,Z 146.209,A -85,B 0,C 180,E1 -21474.076,E2 -21474.076} C_VEL
LIN {X 0,Y 199.652,Z 146.314,A -85,B 0,C 180,E1 -21476.651,E2 -21476.651} C_VEL
LIN {X 0,Y 200.172,Z 148.104,A -85,B 0,C 180,E1 -21477.288,E2 -21477.288} C_VEL
LIN {X 0,Y 201.728,Z 150.422,A -85,B 0,C 180,E1 -21477.988,E2 -21477.988} C_VEL
LIN {X 0,Y 203.125,Z 151.786,A -85,B 0,C 180,E1 -21478.565,E2 -21478.565} C_VEL
LIN {X 0,Y 205.964,Z 155.701,A -85,B 0,C 180,E1 -21479.771,E2 -21479.771} C_VEL
LIN {X 0,Y 212.215,Z 164.821,A -85,B 0,C 180,E1 -21482.252,E2 -21482.252} C_VEL
LIN {X 0,Y 220.091,Z 177.138,A -85,B 0,C 180,E1 -21485.101,E2 -21485.101} C_VEL
LIN {X 0,Y 228.271,Z 191.407,A -85,B 0,C 180,E1 -21487.83,E2 -21487.83} C_VEL
LIN {X 0,Y 236.729,Z 208.424,A -85,B 0,C 180,E1 -21490.461,E2 -21490.461} C_VEL
LIN {X 0,Y 240.979,Z 218.136,A -85,B 0,C 180,E1 -21491.734,E2 -21491.734} C_VEL
LIN {X 0,Y 234.956,Z 314.947,A -85,B 0,C 180,E1 -21494.527,E2 -21494.527} C_VEL
LIN {X 0,Y 233.292,Z 330.271,A -85,B 0,C 180,E1 -21495.233,E2 -21495.233} C_VEL
LIN {X 0,Y 231.074,Z 345.249,A -85,B 0,C 180,E1 -21496.254,E2 -21496.254} C_VEL
LIN {X 0,Y 228.297,Z 359.563,A -85,B 0,C 180,E1 -21497.556,E2 -21497.556} C_VEL
LIN {X 0,Y 225.369,Z 372.012,A -85,B 0,C 180,E1 -21498.989,E2 -21498.989} C_VEL
LIN {X 0,Y 221.832,Z 385.107,A -85,B 0,C 180,E1 -21500.885,E2 -21500.885} C_VEL
LIN {X 0,Y 218.096,Z 397.229,A -85,B 0,C 180,E1 -21503.059,E2 -21503.059} C_VEL
LIN {X 0,Y 214.731,Z 407.453,A -85,B 0,C 180,E1 -21505.307,E2 -21505.307} C_VEL
LIN {X 0,Y 210.955,Z 418.035,A -85,B 0,C 180,E1 -21508.134,E2 -21508.134} C_VEL
LIN {X 0,Y 207.241,Z 428.051,A -85,B 0,C 180,E1 -21511.457,E2 -21511.457} C_VEL
LIN {X 0,Y 203.957,Z 436.776,A -85,B 0,C 180,E1 -21515.097,E2 -21515.097} C_VEL
LIN {X 0,Y 201.248,Z 444.214,A -85,B 0,C 180,E1 -21519.041,E2 -21519.041} C_VEL
LIN {X 0,Y 199.671,Z 448.944,A -85,B 0,C 180,E1 -21522.192,E2 -21522.192} C_VEL
LIN {X 0,Y 198.159,Z 453.936,A -85,B 0,C 180,E1 -21526.483,E2 -21526.483} C_VEL
LIN {X 0,Y 197.144,Z 457.515,A -85,B 0,C 180,E1 -21530.885,E2 -21530.885} C_VEL
LIN {X 0,Y 196.771,Z 459.691,A -85,B 0,C 180,E1 -21535.379,E2 -21535.379} C_VEL
LIN {X 0,Y 196.759,Z 460.256,A -85,B 0,C 180,E1 -21537.668,E2 -21537.668} C_VEL
LIN {X 0,Y 196.996,Z 460.395,A -85,B 0,C 180,E1 -21541.104,E2 -21541.104} C_VEL
LIN {X 0,Y 197.71,Z 459.573,A -85,B 0,C 180,E1 -21545.155,E2 -21545.155} C_VEL
LIN {X 0,Y 199.045,Z 457.451,A -85,B 0,C 180,E1 -21549.461,E2 -21549.461} C_VEL
LIN {X 0,Y 200.505,Z 455.048,A -85,B 0,C 180,E1 -21552.6,E2 -21552.6} C_VEL
LIN {X 0,Y 203.011,Z 450.771,A -85,B 0,C 180,E1 -21556.635,E2 -21556.635} C_VEL
LIN {X 0,Y 206.073,Z 445.58,A -85,B 0,C 180,E1 -21560.292,E2 -21560.292} C_VEL
LIN {X 0,Y 210.343,Z 438.458,A -85,B 0,C 180,E1 -21564.12,E2 -21564.12} C_VEL
LIN {X 0,Y 214.784,Z 430.625,A -85,B 0,C 180,E1 -21567.412,E2 -21567.412} C_VEL
LIN {X 0,Y 219.849,Z 421.145,A -85,B 0,C 180,E1 -21570.567,E2 -21570.567} C_VEL
LIN {X 0,Y 225.163,Z 410.509,A -85,B 0,C 180,E1 -21573.362,E2 -21573.362} C_VEL
LIN {X 0,Y 225.879,Z 409.093,A -85,B 0,C 180,E1 -21573.692,E2 -21573.692} C_VEL
LIN {X 0,Y 225.303,Z 408.299,A -85,B 0,C 180,E1 -21574.105,E2 -21574.105} C_VEL
LIN {X 0,Y 215.848,Z 407.375,A -85,B 0,C 180,E1 -21577,E2 -21577} C_VEL
LIN {X 0,Y 207.777,Z 405.786,A -85,B 0,C 180,E1 -21580.229,E2 -21580.229} C_VEL
LIN {X 0,Y 200.961,Z 403.734,A -85,B 0,C 180,E1 -21583.752,E2 -21583.752} C_VEL
LIN {X 0,Y 199.75,Z 402.468,A -85,B 0,C 180,E1 -21584.829,E2 -21584.829} C_VEL
LIN {X 0,Y 199.754,Z 402.236,A -85,B 0,C 180,E1 -21584.96,E2 -21584.96} C_VEL
LIN {X 0,Y 198.542,Z 412.356,A -85,B 0,C 180,E1 -21588.773,E2 -21588.773} C_VEL
LIN {X 0,Y 198,Z 419.205,A -85,B 0,C 180,E1 -21591.837,E2 -21591.837} C_VEL
LIN {X 0,Y 197.632,Z 426.144,A -85,B 0,C 180,E1 -21595.592,E2 -21595.592} C_VEL
LIN {X 0,Y 197.662,Z 431.256,A -85,B 0,C 180,E1 -21598.981,E2 -21598.981} C_VEL
LIN {X 0,Y 197.888,Z 436.144,A -85,B 0,C 180,E1 -21603.053,E2 -21603.053} C_VEL
LIN {X 0,Y 198.271,Z 438.973,A -85,B 0,C 180,E1 -21606.104,E2 -21606.104} C_VEL
LIN {X 0,Y 199.582,Z 441.764,A -85,B 0,C 180,E1 -21610.14,E2 -21610.14} C_VEL
LIN {X 0,Y 201.687,Z 443.519,A -85,B 0,C 180,E1 -21614.118,E2 -21614.118} C_VEL
LIN {X 0,Y 204.583,Z 444.202,A -85,B 0,C 180,E1 -21618.009,E2 -21618.009} C_VEL
LIN {X 0,Y 208.523,Z 443.899,A -85,B 0,C 180,E1 -21621.761,E2 -21621.761} C_VEL
LIN {X 0,Y 213.289,Z 442.689,A -85,B 0,C 180,E1 -21625.363,E2 -21625.363} C_VEL
LIN {X 0,Y 217.396,Z 441.135,A -85,B 0,C 180,E1 -21627.785,E2 -21627.785} C_VEL
LIN {X 0,Y 219.457,Z 440.211,A -85,B 0,C 180,E1 -21629.216,E2 -21629.216} C_VEL
LIN {X 0,Y 223.414,Z 437.781,A -85,B 0,C 180,E1 -21633.674,E2 -21633.674} C_VEL
LIN {X 0,Y 225.671,Z 436.49,A -85,B 0,C 180,E1 -21635.022,E2 -21635.022} C_VEL
LIN {X 0,Y 226.672,Z 435.951,A -85,B 0,C 180,E1 -21635.427,E2 -21635.427} C_VEL
LIN {X 0,Y 236.453,Z 430.55,A -85,B 0,C 180,E1 -21638.621,E2 -21638.621} C_VEL
LIN {X 0,Y 245.79,Z 424.744,A -85,B 0,C 180,E1 -21641.12,E2 -21641.12} C_VEL
LIN {X 0,Y 255.728,Z 417.825,A -85,B 0,C 180,E1 -21643.397,E2 -21643.397} C_VEL
LIN {X 0,Y 252.376,Z 420.596,A -85,B 0,C 180,E1 -21644.187,E2 -21644.187} C_VEL
LIN {X 0,Y 240.827,Z 429.579,A -85,B 0,C 180,E1 -21646.702,E2 -21646.702} C_VEL
LIN {X 0,Y 231.427,Z 436.428,A -85,B 0,C 180,E1 -21649.238,E2 -21649.238} C_VEL
LIN {X 0,Y 222.078,Z 442.818,A -85,B 0,C 180,E1 -21652.294,E2 -21652.294} C_VEL
LIN {X 0,Y 213.25,Z 448.4,A -85,B 0,C 180,E1 -21655.926,E2 -21655.926} C_VEL
LIN {X 0,Y 206.795,Z 452.212,A -85,B 0,C 180,E1 -21659.351,E2 -21659.351} C_VEL
LIN {X 0,Y 201.39,Z 455.2,A -85,B 0,C 180,E1 -21663.021,E2 -21663.021} C_VEL
LIN {X 0,Y 196.327,Z 457.647,A -85,B 0,C 180,E1 -21667.645,E2 -21667.645} C_VEL
LIN {X 0,Y 193.905,Z 461.837,A -85,B 0,C 180,E1 -21670.962,E2 -21670.962} C_VEL
LIN {X 0,Y 191.849,Z 465.782,A -85,B 0,C 180,E1 -21675.142,E2 -21675.142} C_VEL
LIN {X 0,Y 190.642,Z 468.483,A -85,B 0,C 180,E1 -21679.378,E2 -21679.378} C_VEL
LIN {X 0,Y 190.203,Z 470.011,A -85,B 0,C 180,E1 -21683.636,E2 -21683.636} C_VEL
LIN {X 0,Y 190.178,Z 470.379,A -85,B 0,C 180,E1 -21687.882,E2 -21687.882} C_VEL
LIN {X 0,Y 190.272,Z 470.123,A -85,B 0,C 180,E1 -21690,E2 -21690} C_VEL
LIN {X 0,Y 190.16,Z 468.694,A -85,B 0,C 180,E1 -21694.239,E2 -21694.239} C_VEL
LIN {X 0,Y 190.321,Z 466.012,A -85,B 0,C 180,E1 -21698.494,E2 -21698.494} C_VEL
LIN {X 0,Y 190.98,Z 462.001,A -85,B 0,C 180,E1 -21702.756,E2 -21702.756} C_VEL
LIN {X 0,Y 192.353,Z 457.49,A -85,B 0,C 180,E1 -21706.449,E2 -21706.449} C_VEL
LIN {X 0,Y 195.172,Z 456.737,A -85,B 0,C 180,E1 -21711.106,E2 -21711.106} C_VEL
LIN {X 0,Y 199.017,Z 455.11,A -85,B 0,C 180,E1 -21715.072,E2 -21715.072} C_VEL
LIN {X 0,Y 203.88,Z 452.615,A -85,B 0,C 180,E1 -21718.855,E2 -21718.855} C_VEL
LIN {X 0,Y 211.477,Z 448.226,A -85,B 0,C 180,E1 -21723.253,E2 -21723.253} C_VEL
LIN {X 0,Y 218.732,Z 443.685,A -85,B 0,C 180,E1 -21726.471,E2 -21726.471} C_VEL
LIN {X 0,Y 226.981,Z 438.249,A -85,B 0,C 180,E1 -21729.401,E2 -21729.401} C_VEL
LIN {X 0,Y 238.474,Z 430.044,A -85,B 0,C 180,E1 -21732.674,E2 -21732.674} C_VEL
LIN {X 0,Y 250.44,Z 420.784,A -85,B 0,C 180,E1 -21735.376,E2 -21735.376} C_VEL
LIN {X 0,Y 253.844,Z 417.972,A -85,B 0,C 180,E1 -21736.042,E2 -21736.042} C_VEL
LIN {X 0,Y 255.783,Z 416.347,A -85,B 0,C 180,E1 -21736.614,E2 -21736.614} C_VEL
LIN {X 0,Y 245.75,Z 423.422,A -85,B 0,C 180,E1 -21738.871,E2 -21738.871} C_VEL
LIN {X 0,Y 236.455,Z 429.319,A -85,B 0,C 180,E1 -21741.379,E2 -21741.379} C_VEL
LIN {X 0,Y 227.858,Z 434.219,A -85,B 0,C 180,E1 -21744.125,E2 -21744.125} C_VEL
LIN {X 0,Y 220.154,Z 438.102,A -85,B 0,C 180,E1 -21747.133,E2 -21747.133} C_VEL
LIN {X 0,Y 213.126,Z 440.999,A -85,B 0,C 180,E1 -21750.355,E2 -21750.355} C_VEL
LIN {X 0,Y 206.999,Z 442.948,A -85,B 0,C 180,E1 -21753.809,E2 -21753.809} C_VEL
LIN {X 0,Y 201.921,Z 443.965,A -85,B 0,C 180,E1 -21757.489,E2 -21757.489} C_VEL
LIN {X 0,Y 197.833,Z 443.972,A -85,B 0,C 180,E1 -21761.354,E2 -21761.354} C_VEL
LIN {X 0,Y 194.76,Z 443.017,A -85,B 0,C 180,E1 -21765.369,E2 -21765.369} C_VEL
LIN {X 0,Y 192.531,Z 441.089,A -85,B 0,C 180,E1 -21769.484,E2 -21769.484} C_VEL
LIN {X 0,Y 191.17,Z 438.04,A -85,B 0,C 180,E1 -21773.669,E2 -21773.669} C_VEL
LIN {X 0,Y 190.731,Z 433.866,A -85,B 0,C 180,E1 -21777.889,E2 -21777.889} C_VEL
LIN {X 0,Y 190.573,Z 428.393,A -85,B 0,C 180,E1 -21782.114,E2 -21782.114} C_VEL
LIN {X 0,Y 190.756,Z 421.419,A -85,B 0,C 180,E1 -21786.346,E2 -21786.346} C_VEL
LIN {X 0,Y 191.265,Z 413.896,A -85,B 0,C 180,E1 -21790.052,E2 -21790.052} C_VEL
LIN {X 0,Y 192.157,Z 404.833,A -85,B 0,C 180,E1 -21793.753,E2 -21793.753} C_VEL
LIN {X 0,Y 193.203,Z 395.607,A -85,B 0,C 180,E1 -21796.919,E2 -21796.919} C_VEL
LIN {X 0,Y 194.853,Z 383.773,A -85,B 0,C 180,E1 -21800.319,E2 -21800.319} C_VEL
LIN {X 0,Y 196.874,Z 370.856,A -85,B 0,C 180,E1 -21803.4,E2 -21803.4} C_VEL
LIN {X 0,Y 198.778,Z 358,A -85,B 0,C 180,E1 -21805.947,E2 -21805.947} C_VEL
LIN {X 0,Y 200.858,Z 344.355,A -85,B 0,C 180,E1 -21808.189,E2 -21808.189} C_VEL
LIN {X 0,Y 202.881,Z 329.391,A -85,B 0,C 180,E1 -21810.201,E2 -21810.201} C_VEL
LIN {X 0,Y 204.727,Z 313.979,A -85,B 0,C 180,E1 -21811.858,E2 -21811.858} C_VEL
LIN {X 0,Y 206.318,Z 297.05,A -85,B 0,C 180,E1 -21813.245,E2 -21813.245} C_VEL
LIN {X 0,Y 214.385,Z 200.772,A -85,B 0,C 180,E1 -21818.69,E2 -21818.69} C_VEL
LIN {X 0,Y 213.371,Z 197.725,A -85,B 0,C 180,E1 -21818.973,E2 -21818.973} C_VEL
LIN {X 0,Y 200.638,Z 166.575,A -85,B 0,C 180,E1 -21822.364,E2 -21822.364} C_VEL
LIN {X 0,Y 192.653,Z 147.705,A -85,B 0,C 180,E1 -21824.674,E2 -21824.674} C_VEL
LIN {X 0,Y 192.551,Z 147.089,A -85,B 0,C 180,E1 -21824.834,E2 -21824.834} C_VEL
LIN {X 0,Y 192.508,Z 147.125,A -85,B 0,C 180,E1 -21830.056,E2 -21830.056} C_VEL
LIN {X 0,Y 192.594,Z 147.171,A -85,B 0,C 180,E1 -21834.061,E2 -21834.061} C_VEL
LIN {X 0,Y 192.982,Z 148.784,A -85,B 0,C 180,E1 -21834.523,E2 -21834.523} C_VEL
LIN {X 0,Y 194.455,Z 151.11,A -85,B 0,C 180,E1 -21835.285,E2 -21835.285} C_VEL
LIN {X 0,Y 196.43,Z 152.787,A -85,B 0,C 180,E1 -21836.176,E2 -21836.176} C_VEL
LIN {X 0,Y 198.443,Z 156.044,A -85,B 0,C 180,E1 -21837.143,E2 -21837.143} C_VEL
LIN {X 0,Y 200.423,Z 158.272,A -85,B 0,C 180,E1 -21838,E2 -21838} C_VEL
LIN {X 0,Y 206.487,Z 166.977,A -85,B 0,C 180,E1 -21840.586,E2 -21840.586} C_VEL
LIN {X 0,Y 213.258,Z 177.445,A -85,B 0,C 180,E1 -21843.226,E2 -21843.226} C_VEL
LIN {X 0,Y 219.179,Z 187.435,A -85,B 0,C 180,E1 -21845.364,E2 -21845.364} C_VEL
LIN {X 0,Y 225.577,Z 199.189,A -85,B 0,C 180,E1 -21847.545,E2 -21847.545} C_VEL
LIN {X 0,Y 233.804,Z 216.439,A -85,B 0,C 180,E1 -21850.177,E2 -21850.177} C_VEL
LIN {X 0,Y 235.391,Z 220.172,A -85,B 0,C 180,E1 -21850.675,E2 -21850.675} C_VEL
LIN {X 0,Y 229.295,Z 315.28,A -85,B 0,C 180,E1 -21853.473,E2 -21853.473} C_VEL
LIN {X 0,Y 227.562,Z 330.677,A -85,B 0,C 180,E1 -21854.196,E2 -21854.196} C_VEL
LIN {X 0,Y 225.336,Z 345.302,A -85,B 0,C 180,E1 -21855.211,E2 -21855.211} C_VEL
LIN {X 0,Y 222.472,Z 359.603,A -85,B 0,C 180,E1 -21856.527,E2 -21856.527} C_VEL
LIN {X 0,Y 219.433,Z 372.089,A -85,B 0,C 180,E1 -21857.984,E2 -21857.984} C_VEL
LIN {X 0,Y 215.772,Z 385.204,A -85,B 0,C 180,E1 -21859.917,E2 -21859.917} C_VEL
LIN {X 0,Y 212.097,Z 396.712,A -85,B 0,C 180,E1 -21862.003,E2 -21862.003} C_VEL
LIN {X 0,Y 208.066,Z 408.525,A -85,B 0,C 180,E1 -21864.67,E2 -21864.67} C_VEL
LIN {X 0,Y 203.975,Z 419.437,A -85,B 0,C 180,E1 -21867.728,E2 -21867.728} C_VEL
LIN {X 0,Y 200.33,Z 428.839,A -85,B 0,C 180,E1 -21871.005,E2 -21871.005} C_VEL
LIN {X 0,Y 197.34,Z 436.505,A -85,B 0,C 180,E1 -21874.291,E2 -21874.291} C_VEL
LIN {X 0,Y 194.498,Z 443.962,A -85,B 0,C 180,E1 -21878.31,E2 -21878.31} C_VEL
LIN {X 0,Y 192.339,Z 450.164,A -85,B 0,C 180,E1 -21882.664,E2 -21882.664} C_VEL
LIN {X 0,Y 190.931,Z 454.642,A -85,B 0,C 180,E1 -21886.854,E2 -21886.854} C_VEL
LIN {X 0,Y 190.306,Z 456.709,A -85,B 0,C 180,E1 -21889.413,E2 -21889.413} C_VEL
LIN {X 0,Y 189.71,Z 459.318,A -85,B 0,C 180,E1 -21894.048,E2 -21894.048} C_VEL
LIN {X 0,Y 189.678,Z 460.291,A -85,B 0,C 180,E1 -21897.219,E2 -21897.219} C_VEL
LIN {X 0,Y 189.979,Z 460.572,A -85,B 0,C 180,E1 -21901.694,E2 -21901.694} C_VEL
LIN {X 0,Y 190.82,Z 459.607,A -85,B 0,C 180,E1 -21906.107,E2 -21906.107} C_VEL
LIN {X 0,Y 192.048,Z 457.865,A -85,B 0,C 180,E1 -21909.78,E2 -21909.78} C_VEL
LIN {X 0,Y 194.552,Z 453.951,A -85,B 0,C 180,E1 -21914.783,E2 -21914.783} C_VEL
LIN {X 0,Y 197.204,Z 449.858,A -85,B 0,C 180,E1 -21918.452,E2 -21918.452} C_VEL
LIN {X 0,Y 201.174,Z 443.589,A -85,B 0,C 180,E1 -21922.634,E2 -21922.634} C_VEL
LIN {X 0,Y 205.699,Z 436.39,A -85,B 0,C 180,E1 -21926.28,E2 -21926.28} C_VEL
LIN {X 0,Y 210.296,Z 428.692,A -85,B 0,C 180,E1 -21929.379,E2 -21929.379} C_VEL
LIN {X 0,Y 215.663,Z 418.901,A -85,B 0,C 180,E1 -21932.524,E2 -21932.524} C_VEL
LIN {X 0,Y 218.017,Z 414.549,A -85,B 0,C 180,E1 -21933.688,E2 -21933.688} C_VEL
LIN {X 0,Y 218.13,Z 413.074,A -85,B 0,C 180,E1 -21934.216,E2 -21934.216} C_VEL
LIN {X 0,Y 206.933,Z 411.679,A -85,B 0,C 180,E1 -21938.062,E2 -21938.062} C_VEL
LIN {X 0,Y 196.251,Z 408.86,A -85,B 0,C 180,E1 -21943.351,E2 -21943.351} C_VEL
LIN {X 0,Y 193.236,Z 407.807,A -85,B 0,C 180,E1 -21945.25,E2 -21945.25} C_VEL
LIN {X 0,Y 192.112,Z 406.973,A -85,B 0,C 180,E1 -21946.243,E2 -21946.243} C_VEL
LIN {X 0,Y 192.019,Z 406.448,A -85,B 0,C 180,E1 -21946.641,E2 -21946.641} C_VEL
LIN {X 0,Y 191.178,Z 415.636,A -85,B 0,C 180,E1 -21950.477,E2 -21950.477} C_VEL
LIN {X 0,Y 190.695,Z 423.187,A -85,B 0,C 180,E1 -21954.312,E2 -21954.312} C_VEL
LIN {X 0,Y 190.626,Z 428.979,A -85,B 0,C 180,E1 -21957.886,E2 -21957.886} C_VEL
LIN {X 0,Y 190.756,Z 434.472,A -85,B 0,C 180,E1 -21962.111,E2 -21962.111} C_VEL
LIN {X 0,Y 191.218,Z 438.683,A -85,B 0,C 180,E1 -21966.33,E2 -21966.33} C_VEL
LIN {X 0,Y 192.596,Z 441.764,A -85,B 0,C 180,E1 -21970.512,E2 -21970.512} C_VEL
LIN {X 0,Y 194.797,Z 443.735,A -85,B 0,C 180,E1 -21974.628,E2 -21974.628} C_VEL
LIN {X 0,Y 197.86,Z 444.742,A -85,B 0,C 180,E1 -21978.643,E2 -21978.643} C_VEL
LIN {X 0,Y 201.986,Z 444.779,A -85,B 0,C 180,E1 -21982.503,E2 -21982.503} C_VEL
LIN {X 0,Y 206.979,Z 443.831,A -85,B 0,C 180,E1 -21986.194,E2 -21986.194} C_VEL
LIN {X 0,Y 213.197,Z 441.934,A -85,B 0,C 180,E1 -21989.634,E2 -21989.634} C_VEL
LIN {X 0,Y 220.122,Z 439.105,A -85,B 0,C 180,E1 -21992.872,E2 -21992.872} C_VEL
LIN {X 0,Y 226.672,Z 435.951,A -85,B 0,C 180,E1 -21995.427,E2 -21995.427} C_VEL
LIN {X 0,Y 229.491,Z 434.437,A -85,B 0,C 180,E1 -21996.677,E2 -21996.677} C_VEL
LIN {X 0,Y 236.307,Z 430.574,A -85,B 0,C 180,E1 -22000.617,E2 -22000.617} C_VEL
LIN {X 0,Y 239.985,Z 428.488,A -85,B 0,C 180,E1 -22001.909,E2 -22001.909} C_VEL
LIN {X 0,Y 240.61,Z 428.102,A -85,B 0,C 180,E1 -22002.067,E2 -22002.067} C_VEL
LIN {X 0,Y 245.973,Z 424.885,A -85,B 0,C 180,E1 -22003.293,E2 -22003.293} C_VEL
LIN {X 0,Y 241.981,Z 427.73,A -85,B 0,C 180,E1 -22004.223,E2 -22004.223} C_VEL
LIN {X 0,Y 230.985,Z 435.201,A -85,B 0,C 180,E1 -22006.797,E2 -22006.797} C_VEL
LIN {X 0,Y 219.458,Z 442.406,A -85,B 0,C 180,E1 -22010.172,E2 -22010.172} C_VEL
LIN {X 0,Y 209.313,Z 448.224,A -85,B 0,C 180,E1 -22014.014,E2 -22014.014} C_VEL
LIN {X 0,Y 200.717,Z 452.694,A -85,B 0,C 180,E1 -22018.317,E2 -22018.317} C_VEL
LIN {X 0,Y 195.05,Z 455.269,A -85,B 0,C 180,E1 -22022.069,E2 -22022.069} C_VEL
LIN {X 0,Y 189.982,Z 457.402,A -85,B 0,C 180,E1 -22026.567,E2 -22026.567} C_VEL
LIN {X 0,Y 187.132,Z 461.873,A -85,B 0,C 180,E1 -22030.244,E2 -22030.244} C_VEL
LIN {X 0,Y 184.927,Z 465.758,A -85,B 0,C 180,E1 -22034.572,E2 -22034.572} C_VEL
LIN {X 0,Y 183.601,Z 468.403,A -85,B 0,C 180,E1 -22038.966,E2 -22038.966} C_VEL
LIN {X 0,Y 183.115,Z 469.869,A -85,B 0,C 180,E1 -22043.388,E2 -22043.388} C_VEL
LIN {X 0,Y 183.075,Z 470.177,A -85,B 0,C 180,E1 -22047.8,E2 -22047.8} C_VEL
LIN {X 0,Y 183.177,Z 469.891,A -85,B 0,C 180,E1 -22050,E2 -22050} C_VEL
LIN {X 0,Y 183.072,Z 468.399,A -85,B 0,C 180,E1 -22054.403,E2 -22054.403} C_VEL
LIN {X 0,Y 183.25,Z 465.651,A -85,B 0,C 180,E1 -22058.824,E2 -22058.824} C_VEL
LIN {X 0,Y 183.994,Z 461.573,A -85,B 0,C 180,E1 -22063.249,E2 -22063.249} C_VEL
LIN {X 0,Y 185.557,Z 456.801,A -85,B 0,C 180,E1 -22067.212,E2 -22067.212} C_VEL
LIN {X 0,Y 188.529,Z 456.395,A -85,B 0,C 180,E1 -22071.887,E2 -22071.887} C_VEL
LIN {X 0,Y 192.564,Z 455.081,A -85,B 0,C 180,E1 -22075.974,E2 -22075.974} C_VEL
LIN {X 0,Y 197.677,Z 452.883,A -85,B 0,C 180,E1 -22079.851,E2 -22079.851} C_VEL
LIN {X 0,Y 203.879,Z 449.866,A -85,B 0,C 180,E1 -22083.473,E2 -22083.473} C_VEL
LIN {X 0,Y 211.134,Z 445.963,A -85,B 0,C 180,E1 -22086.81,E2 -22086.81} C_VEL
LIN {X 0,Y 221.684,Z 439.831,A -85,B 0,C 180,E1 -22090.535,E2 -22090.535} C_VEL
LIN {X 0,Y 233.501,Z 432.254,A -85,B 0,C 180,E1 -22093.81,E2 -22093.81} C_VEL
LIN {X 0,Y 243.845,Z 425.12,A -85,B 0,C 180,E1 -22096.099,E2 -22096.099} C_VEL
LIN {X 0,Y 245.943,Z 423.518,A -85,B 0,C 180,E1 -22096.701,E2 -22096.701} C_VEL
LIN {X 0,Y 235.991,Z 429.469,A -85,B 0,C 180,E1 -22099.068,E2 -22099.068} C_VEL
LIN {X 0,Y 224.585,Z 435.457,A -85,B 0,C 180,E1 -22102.395,E2 -22102.395} C_VEL
LIN {X 0,Y 218.314,Z 438.325,A -85,B 0,C 180,E1 -22104.588,E2 -22104.588} C_VEL
LIN {X 0,Y 210.73,Z 441.274,A -85,B 0,C 180,E1 -22107.751,E2 -22107.751} C_VEL
LIN {X 0,Y 203.847,Z 443.378,A -85,B 0,C 180,E1 -22111.14,E2 -22111.14} C_VEL
LIN {X 0,Y 197.937,Z 444.492,A -85,B 0,C 180,E1 -22114.782,E2 -22114.782} C_VEL
LIN {X 0,Y 193.134,Z 444.673,A -85,B 0,C 180,E1 -22118.661,E2 -22118.661} C_VEL
LIN {X 0,Y 189.389,Z 443.941,A -85,B 0,C 180,E1 -22122.731,E2 -22122.731} C_VEL
LIN {X 0,Y 186.6,Z 442.17,A -85,B 0,C 180,E1 -22126.94,E2 -22126.94} C_VEL
LIN {X 0,Y 184.424,Z 438.651,A -85,B 0,C 180,E1 -22132.223,E2 -22132.223} C_VEL
LIN {X 0,Y 183.748,Z 434.392,A -85,B 0,C 180,E1 -22136.712,E2 -22136.712} C_VEL
LIN {X 0,Y 183.522,Z 428.983,A -85,B 0,C 180,E1 -22141.098,E2 -22141.098} C_VEL
LIN {X 0,Y 183.605,Z 422.762,A -85,B 0,C 180,E1 -22145.108,E2 -22145.108} C_VEL
LIN {X 0,Y 184.003,Z 415.835,A -85,B 0,C 180,E1 -22148.789,E2 -22148.789} C_VEL
LIN {X 0,Y 184.746,Z 407.113,A -85,B 0,C 180,E1 -22152.636,E2 -22152.636} C_VEL
LIN {X 0,Y 185.811,Z 398.228,A -85,B 0,C 180,E1 -22155.916,E2 -22155.916} C_VEL
LIN {X 0,Y 187.426,Z 385.921,A -85,B 0,C 180,E1 -22159.724,E2 -22159.724} C_VEL
LIN {X 0,Y 189.361,Z 373.305,A -85,B 0,C 180,E1 -22162.937,E2 -22162.937} C_VEL
LIN {X 0,Y 191.486,Z 359.501,A -85,B 0,C 180,E1 -22165.84,E2 -22165.84} C_VEL
LIN {X 0,Y 193.796,Z 344.492,A -85,B 0,C 180,E1 -22168.424,E2 -22168.424} C_VEL
LIN {X 0,Y 195.934,Z 328.947,A -85,B 0,C 180,E1 -22170.587,E2 -22170.587} C_VEL
LIN {X 0,Y 197.859,Z 312.791,A -85,B 0,C 180,E1 -22172.346,E2 -22172.346} C_VEL
LIN {X 0,Y 199.496,Z 295.431,A -85,B 0,C 180,E1 -22173.777,E2 -22173.777} C_VEL
LIN {X 0,Y 207.584,Z 201.812,A -85,B 0,C 180,E1 -22179.272,E2 -22179.272} C_VEL
LIN {X 0,Y 194.39,Z 169.437,A -85,B 0,C 180,E1 -22182.912,E2 -22182.912} C_VEL
LIN {X 0,Y 185.609,Z 148.693,A -85,B 0,C 180,E1 -22185.544,E2 -22185.544} C_VEL
LIN {X 0,Y 185.475,Z 147.961,A -85,B 0,C 180,E1 -22185.659,E2 -22185.659} C_VEL
LIN {X 0,Y 185.471,Z 148.011,A -85,B 0,C 180,E1 -22191.099,E2 -22191.099} C_VEL
LIN {X 0,Y 186.392,Z 150.655,A -85,B 0,C 180,E1 -22191.731,E2 -22191.731} C_VEL
LIN {X 0,Y 188.219,Z 152.709,A -85,B 0,C 180,E1 -22192.718,E2 -22192.718} C_VEL
LIN {X 0,Y 189.576,Z 153.754,A -85,B 0,C 180,E1 -22193.399,E2 -22193.399} C_VEL
LIN {X 0,Y 191.426,Z 156.863,A -85,B 0,C 180,E1 -22194.42,E2 -22194.42} C_VEL
LIN {X 0,Y 193.494,Z 159.006,A -85,B 0,C 180,E1 -22195.42,E2 -22195.42} C_VEL
LIN {X 0,Y 196.106,Z 162.64,A -85,B 0,C 180,E1 -22196.68,E2 -22196.68} C_VEL
LIN {X 0,Y 197.355,Z 164.238,A -85,B 0,C 180,E1 -22197.25,E2 -22197.25} C_VEL
LIN {X 0,Y 202.518,Z 171.576,A -85,B 0,C 180,E1 -22199.531,E2 -22199.531} C_VEL
LIN {X 0,Y 210.82,Z 184.73,A -85,B 0,C 180,E1 -22202.899,E2 -22202.899} C_VEL
LIN {X 0,Y 219.124,Z 199.547,A -85,B 0,C 180,E1 -22205.943,E2 -22205.943} C_VEL
LIN {X 0,Y 226.683,Z 215.09,A -85,B 0,C 180,E1 -22208.53,E2 -22208.53} C_VEL
LIN {X 0,Y 229.942,Z 222.467,A -85,B 0,C 180,E1 -22209.592,E2 -22209.592} C_VEL
LIN {X 0,Y 223.768,Z 315.101,A -85,B 0,C 180,E1 -22212.345,E2 -22212.345} C_VEL
LIN {X 0,Y 221.967,Z 330.763,A -85,B 0,C 180,E1 -22213.088,E2 -22213.088} C_VEL
LIN {X 0,Y 219.594,Z 345.78,A -85,B 0,C 180,E1 -22214.148,E2 -22214.148} C_VEL
LIN {X 0,Y 216.724,Z 359.644,A -85,B 0,C 180,E1 -22215.444,E2 -22215.444} C_VEL
LIN {X 0,Y 213.571,Z 372.165,A -85,B 0,C 180,E1 -22216.924,E2 -22216.924} C_VEL
LIN {X 0,Y 209.787,Z 385.296,A -85,B 0,C 180,E1 -22218.894,E2 -22218.894} C_VEL
LIN {X 0,Y 205.678,Z 397.675,A -85,B 0,C 180,E1 -22221.204,E2 -22221.204} C_VEL
LIN {X 0,Y 201.439,Z 409.548,A -85,B 0,C 180,E1 -22223.992,E2 -22223.992} C_VEL
LIN {X 0,Y 197.311,Z 420.067,A -85,B 0,C 180,E1 -22227.05,E2 -22227.05} C_VEL
LIN {X 0,Y 193.456,Z 429.618,A -85,B 0,C 180,E1 -22230.52,E2 -22230.52} C_VEL
LIN {X 0,Y 190.112,Z 437.806,A -85,B 0,C 180,E1 -22234.24,E2 -22234.24} C_VEL
LIN {X 0,Y 187.791,Z 443.685,A -85,B 0,C 180,E1 -22237.527,E2 -22237.527} C_VEL
LIN {X 0,Y 185.446,Z 450.013,A -85,B 0,C 180,E1 -22242.031,E2 -22242.031} C_VEL
LIN {X 0,Y 184.233,Z 453.72,A -85,B 0,C 180,E1 -22245.488,E2 -22245.488} C_VEL
LIN {X 0,Y 183.038,Z 457.484,A -85,B 0,C 180,E1 -22250.216,E2 -22250.216} C_VEL
LIN {X 0,Y 182.569,Z 459.842,A -85,B 0,C 180,E1 -22255.052,E2 -22255.052} C_VEL
LIN {X 0,Y 182.585,Z 460.543,A -85,B 0,C 180,E1 -22257.709,E2 -22257.709} C_VEL
LIN {X 0,Y 182.98,Z 460.739,A -85,B 0,C 180,E1 -22262.529,E2 -22262.529} C_VEL
LIN {X 0,Y 184.158,Z 459.477,A -85,B 0,C 180,E1 -22267.633,E2 -22267.633} C_VEL
LIN {X 0,Y 185.278,Z 457.959,A -85,B 0,C 180,E1 -22270.654,E2 -22270.654} C_VEL
LIN {X 0,Y 187.719,Z 454.455,A -85,B 0,C 180,E1 -22275.344,E2 -22275.344} C_VEL
LIN {X 0,Y 190.583,Z 450.378,A -85,B 0,C 180,E1 -22279.197,E2 -22279.197} C_VEL
LIN {X 0,Y 194.017,Z 445.272,A -85,B 0,C 180,E1 -22282.837,E2 -22282.837} C_VEL
LIN {X 0,Y 198.323,Z 438.892,A -85,B 0,C 180,E1 -22286.385,E2 -22286.385} C_VEL
LIN {X 0,Y 203.327,Z 431.122,A -85,B 0,C 180,E1 -22289.783,E2 -22289.783} C_VEL
LIN {X 0,Y 208.907,Z 421.654,A -85,B 0,C 180,E1 -22293.063,E2 -22293.063} C_VEL
LIN {X 0,Y 210.933,Z 418.083,A -85,B 0,C 180,E1 -22294.106,E2 -22294.106} C_VEL
LIN {X 0,Y 210.878,Z 417.605,A -85,B 0,C 180,E1 -22294.325,E2 -22294.325} C_VEL
LIN {X 0,Y 202.083,Z 416.468,A -85,B 0,C 180,E1 -22297.507,E2 -22297.507} C_VEL
LIN {X 0,Y 194.615,Z 414.833,A -85,B 0,C 180,E1 -22301.033,E2 -22301.033} C_VEL
LIN {X 0,Y 185.704,Z 411.714,A -85,B 0,C 180,E1 -22306.875,E2 -22306.875} C_VEL
LIN {X 0,Y 184.497,Z 410.72,A -85,B 0,C 180,E1 -22308.184,E2 -22308.184} C_VEL
LIN {X 0,Y 184.486,Z 410.289,A -85,B 0,C 180,E1 -22308.462,E2 -22308.462} C_VEL
LIN {X 0,Y 183.859,Z 418.576,A -85,B 0,C 180,E1 -22312.311,E2 -22312.311} C_VEL
LIN {X 0,Y 183.553,Z 424.567,A -85,B 0,C 180,E1 -22315.607,E2 -22315.607} C_VEL
LIN {X 0,Y 183.545,Z 429.588,A -85,B 0,C 180,E1 -22318.902,E2 -22318.902} C_VEL
LIN {X 0,Y 183.781,Z 435.03,A -85,B 0,C 180,E1 -22323.288,E2 -22323.288} C_VEL
LIN {X 0,Y 184.484,Z 439.411,A -85,B 0,C 180,E1 -22327.91,E2 -22327.91} C_VEL
LIN {X 0,Y 186.682,Z 442.881,A -85,B 0,C 180,E1 -22333.054,E2 -22333.054} C_VEL
LIN {X 0,Y 189.456,Z 444.694,A -85,B 0,C 180,E1 -22337.263,E2 -22337.263} C_VEL
LIN {X 0,Y 193.164,Z 445.471,A -85,B 0,C 180,E1 -22341.335,E2 -22341.335} C_VEL
LIN {X 0,Y 197.992,Z 445.348,A -85,B 0,C 180,E1 -22345.211,E2 -22345.211} C_VEL
LIN {X 0,Y 203.794,Z 444.29,A -85,B 0,C 180,E1 -22348.868,E2 -22348.868} C_VEL
LIN {X 0,Y 210.651,Z 442.27,A -85,B 0,C 180,E1 -22352.263,E2 -22352.263} C_VEL
LIN {X 0,Y 218.353,Z 439.38,A -85,B 0,C 180,E1 -22355.405,E2 -22355.405} C_VEL
LIN {X 0,Y 229.032,Z 434.43,A -85,B 0,C 180,E1 -22358.98,E2 -22358.98} C_VEL
LIN {X 0,Y 240.61,Z 428.102,A -85,B 0,C 180,E1 -22362.067,E2 -22362.067} C_VEL
LIN {X 0,Y 239.311,Z 428.934,A -85,B 0,C 180,E1 -22362.106,E2 -22362.106} C_VEL
LIN {X 0,Y 234.79,Z 431.502,A -85,B 0,C 180,E1 -22361.624,E2 -22361.624} C_VEL
LIN {X 0,Y 224.709,Z 436.498,A -85,B 0,C 180,E1 -22359.88,E2 -22359.88} C_VEL
LIN {X 0,Y 218.617,Z 439.12,A -85,B 0,C 180,E1 -22358.423,E2 -22358.423} C_VEL
LIN {X 0,Y 216.798,Z 439.813,A -85,B 0,C 180,E1 -22357.857,E2 -22357.857} C_VEL
LIN {X 0,Y 208.722,Z 442.669,A -85,B 0,C 180,E1 -22354.918,E2 -22354.918} C_VEL
LIN {X 0,Y 201.236,Z 444.764,A -85,B 0,C 180,E1 -22351.591,E2 -22351.591} C_VEL
LIN {X 0,Y 194.479,Z 445.929,A -85,B 0,C 180,E1 -22348.02,E2 -22348.02} C_VEL
LIN {X 0,Y 189.024,Z 446.211,A -85,B 0,C 180,E1 -22344.14,E2 -22344.14} C_VEL
LIN {X 0,Y 184.484,Z 445.545,A -85,B 0,C 180,E1 -22340.05,E2 -22340.05} C_VEL
LIN {X 0,Y 181.106,Z 443.947,A -85,B 0,C 180,E1 -22335.761,E2 -22335.761} C_VEL
LIN {X 0,Y 178.656,Z 441.413,A -85,B 0,C 180,E1 -22331.343,E2 -22331.343} C_VEL
LIN {X 0,Y 176.981,Z 436.711,A -85,B 0,C 180,E1 -22325.697,E2 -22325.697} C_VEL
LIN {X 0,Y 176.535,Z 431.654,A -85,B 0,C 180,E1 -22321.14,E2 -22321.14} C_VEL
LIN {X 0,Y 176.511,Z 426.912,A -85,B 0,C 180,E1 -22317.717,E2 -22317.717} C_VEL
LIN {X 0,Y 176.719,Z 419.242,A -85,B 0,C 180,E1 -22313.147,E2 -22313.147} C_VEL
LIN {X 0,Y 177.076,Z 414.048,A -85,B 0,C 180,E1 -22310.504,E2 -22310.504} C_VEL
LIN {X 0,Y 177.279,Z 414.914,A -85,B 0,C 180,E1 -22309.723,E2 -22309.723} C_VEL
LIN {X 0,Y 186.339,Z 418.518,A -85,B 0,C 180,E1 -22302.438,E2 -22302.438} C_VEL
LIN {X 0,Y 197.074,Z 421.066,A -85,B 0,C 180,E1 -22296.903,E2 -22296.903} C_VEL
LIN {X 0,Y 201.308,Z 421.68,A -85,B 0,C 180,E1 -22295.232,E2 -22295.232} C_VEL
LIN {X 0,Y 203.073,Z 422.82,A -85,B 0,C 180,E1 -22294.134,E2 -22294.134} C_VEL
LIN {X 0,Y 197.27,Z 432.108,A -85,B 0,C 180,E1 -22290.789,E2 -22290.789} C_VEL
LIN {X 0,Y 192.044,Z 439.727,A -85,B 0,C 180,E1 -22287.32,E2 -22287.32} C_VEL
LIN {X 0,Y 187.741,Z 445.705,A -85,B 0,C 180,E1 -22283.862,E2 -22283.862} C_VEL
LIN {X 0,Y 183.874,Z 451.039,A -85,B 0,C 180,E1 -22279.857,E2 -22279.857} C_VEL
LIN {X 0,Y 180.655,Z 455.303,A -85,B 0,C 180,E1 -22275.552,E2 -22275.552} C_VEL
LIN {X 0,Y 178.547,Z 458.055,A -85,B 0,C 180,E1 -22271.592,E2 -22271.592} C_VEL
LIN {X 0,Y 176.738,Z 460.217,A -85,B 0,C 180,E1 -22266.618,E2 -22266.618} C_VEL
LIN {X 0,Y 175.96,Z 460.931,A -85,B 0,C 180,E1 -22262.989,E2 -22262.989} C_VEL
LIN {X 0,Y 175.492,Z 460.788,A -85,B 0,C 180,E1 -22258.23,E2 -22258.23} C_VEL
LIN {X 0,Y 175.537,Z 459.461,A -85,B 0,C 180,E1 -22253.601,E2 -22253.601} C_VEL
LIN {X 0,Y 176.251,Z 456.665,A -85,B 0,C 180,E1 -22248.602,E2 -22248.602} C_VEL
LIN {X 0,Y 177.691,Z 452.455,A -85,B 0,C 180,E1 -22243.728,E2 -22243.728} C_VEL
LIN {X 0,Y 179.744,Z 446.791,A -85,B 0,C 180,E1 -22238.998,E2 -22238.998} C_VEL
LIN {X 0,Y 182.706,Z 439.505,A -85,B 0,C 180,E1 -22234.412,E2 -22234.412} C_VEL
LIN {X 0,Y 186.011,Z 431.646,A -85,B 0,C 180,E1 -22230.541,E2 -22230.541} C_VEL
LIN {X 0,Y 190.049,Z 422.15,A -85,B 0,C 180,E1 -22226.835,E2 -22226.835} C_VEL
LIN {X 0,Y 194.094,Z 412.341,A -85,B 0,C 180,E1 -22223.764,E2 -22223.764} C_VEL
LIN {X 0,Y 198.676,Z 400.288,A -85,B 0,C 180,E1 -22220.738,E2 -22220.738} C_VEL
LIN {X 0,Y 202.985,Z 387.888,A -85,B 0,C 180,E1 -22218.263,E2 -22218.263} C_VEL
LIN {X 0,Y 206.877,Z 375.239,A -85,B 0,C 180,E1 -22216.243,E2 -22216.243} C_VEL
LIN {X 0,Y 210.538,Z 361.497,A -85,B 0,C 180,E1 -22214.511,E2 -22214.511} C_VEL
LIN {X 0,Y 213.864,Z 346.357,A -85,B 0,C 180,E1 -22213.051,E2 -22213.051} C_VEL
LIN {X 0,Y 216.199,Z 332.113,A -85,B 0,C 180,E1 -22212.012,E2 -22212.012} C_VEL
LIN {X 0,Y 218.065,Z 317.003,A -85,B 0,C 180,E1 -22211.26,E2 -22211.26} C_VEL
LIN {X 0,Y 221.551,Z 268.09,A -85,B 0,C 180,E1 -22209.75,E2 -22209.75} C_VEL
LIN {X 0,Y 224.479,Z 224.591,A -85,B 0,C 180,E1 -22208.448,E2 -22208.448} C_VEL
LIN {X 0,Y 216.926,Z 208.207,A -85,B 0,C 180,E1 -22205.79,E2 -22205.79} C_VEL
LIN {X 0,Y 210.707,Z 196.416,A -85,B 0,C 180,E1 -22203.486,E2 -22203.486} C_VEL
LIN {X 0,Y 204.583,Z 185.757,A -85,B 0,C 180,E1 -22201.028,E2 -22201.028} C_VEL
LIN {X 0,Y 197.035,Z 173.905,A -85,B 0,C 180,E1 -22197.734,E2 -22197.734} C_VEL
LIN {X 0,Y 192.883,Z 168.268,A -85,B 0,C 180,E1 -22195.787,E2 -22195.787} C_VEL
LIN {X 0,Y 189.775,Z 164.008,A -85,B 0,C 180,E1 -22194.21,E2 -22194.21} C_VEL
LIN {X 0,Y 187.222,Z 160.808,A -85,B 0,C 180,E1 -22192.859,E2 -22192.859} C_VEL
LIN {X 0,Y 186.364,Z 159.487,A -85,B 0,C 180,E1 -22192.368,E2 -22192.368} C_VEL
LIN {X 0,Y 183.828,Z 156.916,A -85,B 0,C 180,E1 -22190.988,E2 -22190.988} C_VEL
LIN {X 0,Y 182.434,Z 154.423,A -85,B 0,C 180,E1 -22190.104,E2 -22190.104} C_VEL
LIN {X 0,Y 179.935,Z 152.445,A -85,B 0,C 180,E1 -22188.636,E2 -22188.636} C_VEL
LIN {X 0,Y 178.682,Z 150.148,A -85,B 0,C 180,E1 -22187.747,E2 -22187.747} C_VEL
LIN {X 0,Y 178.401,Z 148.84,A -85,B 0,C 180,E1 -22187.443,E2 -22187.443} C_VEL
LIN {X 0,Y 178.407,Z 148.859,A -85,B 0,C 180,E1 -22186.56,E2 -22186.56} C_VEL
LIN {X 0,Y 180.267,Z 153.692,A -85,B 0,C 180,E1 -22185.913,E2 -22185.913} C_VEL
LIN {X 0,Y 192.255,Z 182.221,A -85,B 0,C 180,E1 -22182.247,E2 -22182.247} C_VEL
LIN {X 0,Y 200.63,Z 203.126,A -85,B 0,C 180,E1 -22179.876,E2 -22179.876} C_VEL
LIN {X 0,Y 195.036,Z 266.318,A -85,B 0,C 180,E1 -22176.082,E2 -22176.082} C_VEL
LIN {X 0,Y 192.173,Z 299.703,A -85,B 0,C 180,E1 -22173.899,E2 -22173.899} C_VEL
LIN {X 0,Y 190.548,Z 316.171,A -85,B 0,C 180,E1 -22172.378,E2 -22172.378} C_VEL
LIN {X 0,Y 188.526,Z 331.798,A -85,B 0,C 180,E1 -22170.526,E2 -22170.526} C_VEL
LIN {X 0,Y 186.273,Z 347.759,A -85,B 0,C 180,E1 -22168.14,E2 -22168.14} C_VEL
LIN {X 0,Y 183.991,Z 362.247,A -85,B 0,C 180,E1 -22165.451,E2 -22165.451} C_VEL
LIN {X 0,Y 181.762,Z 376.213,A -85,B 0,C 180,E1 -22162.275,E2 -22162.275} C_VEL
LIN {X 0,Y 179.88,Z 388.785,A -85,B 0,C 180,E1 -22158.805,E2 -22158.805} C_VEL
LIN {X 0,Y 178.403,Z 400.632,A -85,B 0,C 180,E1 -22154.837,E2 -22154.837} C_VEL
LIN {X 0,Y 177.266,Z 410.46,A -85,B 0,C 180,E1 -22150.856,E2 -22150.856} C_VEL
LIN {X 0,Y 176.722,Z 418.656,A -85,B 0,C 180,E1 -22146.853,E2 -22146.853} C_VEL
LIN {X 0,Y 176.459,Z 424.57,A -85,B 0,C 180,E1 -22143.426,E2 -22143.426} C_VEL
LIN {X 0,Y 176.497,Z 429.496,A -85,B 0,C 180,E1 -22140.001,E2 -22140.001} C_VEL
LIN {X 0,Y 176.82,Z 434.887,A -85,B 0,C 180,E1 -22135.441,E2 -22135.441} C_VEL
LIN {X 0,Y 177.735,Z 439.035,A -85,B 0,C 180,E1 -22130.9,E2 -22130.9} C_VEL
LIN {X 0,Y 179.682,Z 442.084,A -85,B 0,C 180,E1 -22126.428,E2 -22126.428} C_VEL
LIN {X 0,Y 182.618,Z 444.1,A -85,B 0,C 180,E1 -22122.069,E2 -22122.069} C_VEL
LIN {X 0,Y 186.555,Z 445.2,A -85,B 0,C 180,E1 -22117.87,E2 -22117.87} C_VEL
LIN {X 0,Y 191.595,Z 445.322,A -85,B 0,C 180,E1 -22113.885,E2 -22113.885} C_VEL
